LIN {X 0,Y 466.661,Z 585.899,A -85,B 0,C 180,E1 -7456.944,E2 -7456.944} C_VEL
LIN {X 0,Y 466.788,Z 583.643,A -85,B 0,C 180,E1 -7458.141,E2 -7458.141} C_VEL
LIN {X 0,Y 466.923,Z 579.745,A -85,B 0,C 180,E1 -7459.594,E2 -7459.594} C_VEL
LIN {X 0,Y 467.085,Z 575.044,A -85,B 0,C 180,E1 -7460.91,E2 -7460.91} C_VEL
LIN {X 0,Y 467.42,Z 568.051,A -85,B 0,C 180,E1 -7462.424,E2 -7462.424} C_VEL
LIN {X 0,Y 467.776,Z 560.313,A -85,B 0,C 180,E1 -7463.747,E2 -7463.747} C_VEL
LIN {X 0,Y 468.215,Z 550.713,A -85,B 0,C 180,E1 -7465.049,E2 -7465.049} C_VEL
LIN {X 0,Y 468.714,Z 540.809,A -85,B 0,C 180,E1 -7466.131,E2 -7466.131} C_VEL
LIN {X 0,Y 469.163,Z 529.664,A -85,B 0,C 180,E1 -7467.102,E2 -7467.102} C_VEL
LIN {X 0,Y 469.668,Z 518.712,A -85,B 0,C 180,E1 -7467.856,E2 -7467.856} C_VEL
LIN {X 0,Y 470.068,Z 506.643,A -85,B 0,C 180,E1 -7468.501,E2 -7468.501} C_VEL
LIN {X 0,Y 470.446,Z 493.985,A -85,B 0,C 180,E1 -7468.984,E2 -7468.984} C_VEL
LIN {X 0,Y 470.619,Z 481.549,A -85,B 0,C 180,E1 -7469.291,E2 -7469.291} C_VEL
LIN {X 0,Y 471.254,Z 391.992,A -85,B 0,C 180,E1 -7470.675,E2 -7470.675} C_VEL
LIN {X 0,Y 468.455,Z 378.274,A -85,B 0,C 180,E1 -7470.994,E2 -7470.994} C_VEL
LIN {X 0,Y 468.774,Z 369.227,A -85,B 0,C 180,E1 -7473.008,E2 -7473.008} C_VEL
LIN {X 0,Y 467.628,Z 363.237,A -85,B 0,C 180,E1 -7474.471,E2 -7474.471} C_VEL
LIN {X 0,Y 467.667,Z 363.231,A -85,B 0,C 180,E1 -7476.905,E2 -7476.905} C_VEL
LIN {X 0,Y 467.668,Z 363.233,A -85,B 0,C 180,E1 -7479.515,E2 -7479.515} C_VEL
LIN {X 0,Y 467.659,Z 363.227,A -85,B 0,C 180,E1 -7482.357,E2 -7482.357} C_VEL
LIN {X 0,Y 467.654,Z 363.229,A -85,B 0,C 180,E1 -7485.885,E2 -7485.885} C_VEL
LIN {X 0,Y 467.627,Z 363.239,A -85,B 0,C 180,E1 -7489.307,E2 -7489.307} C_VEL
LIN {X 0,Y 467.54,Z 363.242,A -85,B 0,C 180,E1 -7492.073,E2 -7492.073} C_VEL
LIN {X 0,Y 467.607,Z 363.237,A -85,B 0,C 180,E1 -7494.886,E2 -7494.886} C_VEL
LIN {X 0,Y 467.622,Z 363.233,A -85,B 0,C 180,E1 -7497.768,E2 -7497.768} C_VEL
LIN {X 0,Y 467.577,Z 363.243,A -85,B 0,C 180,E1 -7501.046,E2 -7501.046} C_VEL
LIN {X 0,Y 467.591,Z 363.235,A -85,B 0,C 180,E1 -7504.242,E2 -7504.242} C_VEL
LIN {X 0,Y 467.551,Z 363.247,A -85,B 0,C 180,E1 -7507.186,E2 -7507.186} C_VEL
LIN {X 0,Y 467.577,Z 363.237,A -85,B 0,C 180,E1 -7510.264,E2 -7510.264} C_VEL
LIN {X 0,Y 467.585,Z 363.238,A -85,B 0,C 180,E1 -7512.566,E2 -7512.566} C_VEL
LIN {X 0,Y 467.569,Z 363.246,A -85,B 0,C 180,E1 -7515.052,E2 -7515.052} C_VEL
LIN {X 0,Y 467.586,Z 363.238,A -85,B 0,C 180,E1 -7517.439,E2 -7517.439} C_VEL
LIN {X 0,Y 467.581,Z 363.243,A -85,B 0,C 180,E1 -7520.855,E2 -7520.855} C_VEL
LIN {X 0,Y 467.558,Z 363.24,A -85,B 0,C 180,E1 -7524.259,E2 -7524.259} C_VEL
LIN {X 0,Y 467.577,Z 363.24,A -85,B 0,C 180,E1 -7527.32,E2 -7527.32} C_VEL
LIN {X 0,Y 467.564,Z 363.244,A -85,B 0,C 180,E1 -7530.666,E2 -7530.666} C_VEL
LIN {X 0,Y 467.621,Z 363.235,A -85,B 0,C 180,E1 -7533.2,E2 -7533.2} C_VEL
LIN {X 0,Y 467.586,Z 363.24,A -85,B 0,C 180,E1 -7536.467,E2 -7536.467} C_VEL
LIN {X 0,Y 467.616,Z 363.232,A -85,B 0,C 180,E1 -7539.777,E2 -7539.777} C_VEL
LIN {X 0,Y 467.602,Z 363.239,A -85,B 0,C 180,E1 -7542.506,E2 -7542.506} C_VEL
LIN {X 0,Y 467.598,Z 363.236,A -85,B 0,C 180,E1 -7545.196,E2 -7545.196} C_VEL
LIN {X 0,Y 467.648,Z 363.228,A -85,B 0,C 180,E1 -7547.854,E2 -7547.854} C_VEL
LIN {X 0,Y 467.674,Z 363.225,A -85,B 0,C 180,E1 -7551.357,E2 -7551.357} C_VEL
LIN {X 0,Y 467.738,Z 363.218,A -85,B 0,C 180,E1 -7553.962,E2 -7553.962} C_VEL
LIN {X 0,Y 467.852,Z 363.203,A -85,B 0,C 180,E1 -7557.417,E2 -7557.417} C_VEL
LIN {X 0,Y 467.873,Z 363.202,A -85,B 0,C 180,E1 -7560,E2 -7560} C_VEL
LIN {X 0,Y 467.851,Z 363.21,A -85,B 0,C 180,E1 -7562.583,E2 -7562.583} C_VEL
LIN {X 0,Y 467.734,Z 363.22,A -85,B 0,C 180,E1 -7566.037,E2 -7566.037} C_VEL
LIN {X 0,Y 467.673,Z 363.23,A -85,B 0,C 180,E1 -7568.643,E2 -7568.643} C_VEL
LIN {X 0,Y 467.647,Z 363.233,A -85,B 0,C 180,E1 -7572.146,E2 -7572.146} C_VEL
LIN {X 0,Y 467.657,Z 363.229,A -85,B 0,C 180,E1 -7575.893,E2 -7575.893} C_VEL
LIN {X 0,Y 467.615,Z 363.232,A -85,B 0,C 180,E1 -7579.308,E2 -7579.308} C_VEL
LIN {X 0,Y 467.528,Z 363.248,A -85,B 0,C 180,E1 -7582.074,E2 -7582.074} C_VEL
LIN {X 0,Y 467.595,Z 363.236,A -85,B 0,C 180,E1 -7584.888,E2 -7584.888} C_VEL
LIN {X 0,Y 467.621,Z 363.234,A -85,B 0,C 180,E1 -7587.769,E2 -7587.769} C_VEL
LIN {X 0,Y 467.565,Z 363.238,A -85,B 0,C 180,E1 -7591.046,E2 -7591.046} C_VEL
LIN {X 0,Y 467.584,Z 363.243,A -85,B 0,C 180,E1 -7594.243,E2 -7594.243} C_VEL
LIN {X 0,Y 467.546,Z 363.241,A -85,B 0,C 180,E1 -7597.188,E2 -7597.188} C_VEL
LIN {X 0,Y 467.592,Z 363.241,A -85,B 0,C 180,E1 -7600.263,E2 -7600.263} C_VEL
LIN {X 0,Y 467.614,Z 363.234,A -85,B 0,C 180,E1 -7602.572,E2 -7602.572} C_VEL
LIN {X 0,Y 467.566,Z 363.238,A -85,B 0,C 180,E1 -7605.054,E2 -7605.054} C_VEL
LIN {X 0,Y 467.585,Z 363.238,A -85,B 0,C 180,E1 -7607.441,E2 -7607.441} C_VEL
LIN {X 0,Y 467.621,Z 363.231,A -85,B 0,C 180,E1 -7610.86,E2 -7610.86} C_VEL
LIN {X 0,Y 467.561,Z 363.243,A -85,B 0,C 180,E1 -7614.261,E2 -7614.261} C_VEL
LIN {X 0,Y 467.581,Z 363.238,A -85,B 0,C 180,E1 -7617.321,E2 -7617.321} C_VEL
LIN {X 0,Y 467.578,Z 363.242,A -85,B 0,C 180,E1 -7620.666,E2 -7620.666} C_VEL
LIN {X 0,Y 467.666,Z 363.405,A -85,B 0,C 180,E1 -7623.445,E2 -7623.445} C_VEL
LIN {X 0,Y 470.093,Z 376.061,A -85,B 0,C 180,E1 -7625.779,E2 -7625.779} C_VEL
LIN {X 0,Y 469.334,Z 392.226,A -85,B 0,C 180,E1 -7628.532,E2 -7628.532} C_VEL
LIN {X 0,Y 468.677,Z 409.488,A -85,B 0,C 180,E1 -7631.437,E2 -7631.437} C_VEL
LIN {X 0,Y 468.279,Z 418.901,A -85,B 0,C 180,E1 -7633.007,E2 -7633.007} C_VEL
LIN {X 0,Y 471.13,Z 438.244,A -85,B 0,C 180,E1 -7633.413,E2 -7633.413} C_VEL
LIN {X 0,Y 470.44,Z 528.202,A -85,B 0,C 180,E1 -7634.817,E2 -7634.817} C_VEL
LIN {X 0,Y 470.054,Z 541.256,A -85,B 0,C 180,E1 -7635.193,E2 -7635.193} C_VEL
LIN {X 0,Y 469.629,Z 553.327,A -85,B 0,C 180,E1 -7635.705,E2 -7635.705} C_VEL
LIN {X 0,Y 469.159,Z 564.727,A -85,B 0,C 180,E1 -7636.354,E2 -7636.354} C_VEL
LIN {X 0,Y 468.609,Z 576.235,A -85,B 0,C 180,E1 -7637.2,E2 -7637.2} C_VEL
LIN {X 0,Y 468.208,Z 587.031,A -85,B 0,C 180,E1 -7638.199,E2 -7638.199} C_VEL
LIN {X 0,Y 467.767,Z 595.658,A -85,B 0,C 180,E1 -7639.175,E2 -7639.175} C_VEL
LIN {X 0,Y 467.397,Z 603.616,A -85,B 0,C 180,E1 -7640.261,E2 -7640.261} C_VEL
LIN {X 0,Y 467.103,Z 611.392,A -85,B 0,C 180,E1 -7641.565,E2 -7641.565} C_VEL
LIN {X 0,Y 466.858,Z 618.538,A -85,B 0,C 180,E1 -7643.083,E2 -7643.083} C_VEL
LIN {X 0,Y 466.762,Z 623.297,A -85,B 0,C 180,E1 -7644.384,E2 -7644.384} C_VEL
LIN {X 0,Y 466.658,Z 626.931,A -85,B 0,C 180,E1 -7645.682,E2 -7645.682} C_VEL
LIN {X 0,Y 466.697,Z 628.81,A -85,B 0,C 180,E1 -7646.547,E2 -7646.547} C_VEL
LIN {X 0,Y 466.68,Z 630.217,A -85,B 0,C 180,E1 -7647.411,E2 -7647.411} C_VEL
LIN {X 0,Y 466.661,Z 631.218,A -85,B 0,C 180,E1 -7648.274,E2 -7648.274} C_VEL
LIN {X 0,Y 466.6,Z 632.044,A -85,B 0,C 180,E1 -7650,E2 -7650} C_VEL
LIN {X 0,Y 466.62,Z 631.827,A -85,B 0,C 180,E1 -7650.863,E2 -7650.863} C_VEL
LIN {X 0,Y 466.661,Z 631.216,A -85,B 0,C 180,E1 -7651.726,E2 -7651.726} C_VEL
LIN {X 0,Y 466.68,Z 630.212,A -85,B 0,C 180,E1 -7652.589,E2 -7652.589} C_VEL
LIN {X 0,Y 466.697,Z 628.807,A -85,B 0,C 180,E1 -7653.453,E2 -7653.453} C_VEL
LIN {X 0,Y 466.69,Z 625.849,A -85,B 0,C 180,E1 -7654.751,E2 -7654.751} C_VEL
LIN {X 0,Y 466.751,Z 621.85,A -85,B 0,C 180,E1 -7656.05,E2 -7656.05} C_VEL
LIN {X 0,Y 466.942,Z 615.716,A -85,B 0,C 180,E1 -7657.568,E2 -7657.568} C_VEL
LIN {X 0,Y 467.15,Z 609.018,A -85,B 0,C 180,E1 -7658.87,E2 -7658.87} C_VEL
LIN {X 0,Y 467.494,Z 600.717,A -85,B 0,C 180,E1 -7660.174,E2 -7660.174} C_VEL
LIN {X 0,Y 467.967,Z 592.229,A -85,B 0,C 180,E1 -7661.258,E2 -7661.258} C_VEL
LIN {X 0,Y 468.439,Z 582.273,A -85,B 0,C 180,E1 -7662.296,E2 -7662.296} C_VEL
LIN {X 0,Y 468.875,Z 571.396,A -85,B 0,C 180,E1 -7663.213,E2 -7663.213} C_VEL
LIN {X 0,Y 469.435,Z 560.072,A -85,B 0,C 180,E1 -7663.969,E2 -7663.969} C_VEL
LIN {X 0,Y 469.907,Z 548.54,A -85,B 0,C 180,E1 -7664.563,E2 -7664.563} C_VEL
LIN {X 0,Y 470.36,Z 535.317,A -85,B 0,C 180,E1 -7665.047,E2 -7665.047} C_VEL
LIN {X 0,Y 470.643,Z 522.537,A -85,B 0,C 180,E1 -7665.342,E2 -7665.342} C_VEL
LIN {X 0,Y 471.202,Z 437.855,A -85,B 0,C 180,E1 -7666.654,E2 -7666.654} C_VEL
LIN {X 0,Y 468.339,Z 418.514,A -85,B 0,C 180,E1 -7667.095,E2 -7667.095} C_VEL
LIN {X 0,Y 469.097,Z 400.424,A -85,B 0,C 180,E1 -7670.156,E2 -7670.156} C_VEL
LIN {X 0,Y 469.966,Z 381.889,A -85,B 0,C 180,E1 -7673.346,E2 -7673.346} C_VEL
LIN {X 0,Y 470.14,Z 375.734,A -85,B 0,C 180,E1 -7674.428,E2 -7674.428} C_VEL
LIN {X 0,Y 467.686,Z 363.229,A -85,B 0,C 180,E1 -7676.851,E2 -7676.851} C_VEL
LIN {X 0,Y 467.587,Z 363.241,A -85,B 0,C 180,E1 -7679.735,E2 -7679.735} C_VEL
LIN {X 0,Y 467.582,Z 363.238,A -85,B 0,C 180,E1 -7682.758,E2 -7682.758} C_VEL
LIN {X 0,Y 467.555,Z 363.248,A -85,B 0,C 180,E1 -7685.889,E2 -7685.889} C_VEL
LIN {X 0,Y 467.621,Z 363.231,A -85,B 0,C 180,E1 -7689.14,E2 -7689.14} C_VEL
LIN {X 0,Y 467.582,Z 363.237,A -85,B 0,C 180,E1 -7692.566,E2 -7692.566} C_VEL
LIN {X 0,Y 467.566,Z 363.239,A -85,B 0,C 180,E1 -7695.052,E2 -7695.052} C_VEL
LIN {X 0,Y 467.619,Z 363.236,A -85,B 0,C 180,E1 -7697.443,E2 -7697.443} C_VEL
LIN {X 0,Y 467.613,Z 363.233,A -85,B 0,C 180,E1 -7700.858,E2 -7700.858} C_VEL
LIN {X 0,Y 467.557,Z 363.243,A -85,B 0,C 180,E1 -7704.26,E2 -7704.26} C_VEL
LIN {X 0,Y 467.576,Z 363.238,A -85,B 0,C 180,E1 -7707.32,E2 -7707.32} C_VEL
LIN {X 0,Y 467.57,Z 363.236,A -85,B 0,C 180,E1 -7710.665,E2 -7710.665} C_VEL
LIN {X 0,Y 467.62,Z 363.234,A -85,B 0,C 180,E1 -7713.2,E2 -7713.2} C_VEL
LIN {X 0,Y 467.584,Z 363.237,A -85,B 0,C 180,E1 -7716.468,E2 -7716.468} C_VEL
LIN {X 0,Y 467.615,Z 363.239,A -85,B 0,C 180,E1 -7719.777,E2 -7719.777} C_VEL
LIN {X 0,Y 467.6,Z 363.23,A -85,B 0,C 180,E1 -7722.507,E2 -7722.507} C_VEL
LIN {X 0,Y 467.6,Z 363.238,A -85,B 0,C 180,E1 -7725.196,E2 -7725.196} C_VEL
LIN {X 0,Y 467.647,Z 363.23,A -85,B 0,C 180,E1 -7727.854,E2 -7727.854} C_VEL
LIN {X 0,Y 467.673,Z 363.23,A -85,B 0,C 180,E1 -7731.357,E2 -7731.357} C_VEL
LIN {X 0,Y 467.735,Z 363.219,A -85,B 0,C 180,E1 -7733.963,E2 -7733.963} C_VEL
LIN {X 0,Y 467.852,Z 363.205,A -85,B 0,C 180,E1 -7737.417,E2 -7737.417} C_VEL
LIN {X 0,Y 467.873,Z 363.202,A -85,B 0,C 180,E1 -7740,E2 -7740} C_VEL
LIN {X 0,Y 467.853,Z 363.199,A -85,B 0,C 180,E1 -7742.583,E2 -7742.583} C_VEL
LIN {X 0,Y 467.739,Z 363.216,A -85,B 0,C 180,E1 -7746.038,E2 -7746.038} C_VEL
LIN {X 0,Y 467.674,Z 363.225,A -85,B 0,C 180,E1 -7748.643,E2 -7748.643} C_VEL
LIN {X 0,Y 467.648,Z 363.224,A -85,B 0,C 180,E1 -7752.146,E2 -7752.146} C_VEL
LIN {X 0,Y 467.631,Z 363.229,A -85,B 0,C 180,E1 -7755.696,E2 -7755.696} C_VEL
LIN {X 0,Y 467.61,Z 363.238,A -85,B 0,C 180,E1 -7758.765,E2 -7758.765} C_VEL
LIN {X 0,Y 467.603,Z 363.24,A -85,B 0,C 180,E1 -7761.278,E2 -7761.278} C_VEL
LIN {X 0,Y 467.568,Z 363.235,A -85,B 0,C 180,E1 -7763.944,E2 -7763.944} C_VEL
LIN {X 0,Y 467.622,Z 363.238,A -85,B 0,C 180,E1 -7766.8,E2 -7766.8} C_VEL
LIN {X 0,Y 467.548,Z 363.241,A -85,B 0,C 180,E1 -7769.739,E2 -7769.739} C_VEL
LIN {X 0,Y 467.579,Z 363.243,A -85,B 0,C 180,E1 -7772.759,E2 -7772.759} C_VEL
LIN {X 0,Y 467.552,Z 363.241,A -85,B 0,C 180,E1 -7775.89,E2 -7775.89} C_VEL
LIN {X 0,Y 467.609,Z 363.237,A -85,B 0,C 180,E1 -7779.143,E2 -7779.143} C_VEL
LIN {X 0,Y 467.616,Z 363.234,A -85,B 0,C 180,E1 -7782.572,E2 -7782.572} C_VEL
LIN {X 0,Y 467.565,Z 363.242,A -85,B 0,C 180,E1 -7786.178,E2 -7786.178} C_VEL
LIN {X 0,Y 467.581,Z 363.244,A -85,B 0,C 180,E1 -7788.724,E2 -7788.724} C_VEL
LIN {X 0,Y 467.567,Z 363.247,A -85,B 0,C 180,E1 -7791.957,E2 -7791.957} C_VEL
LIN {X 0,Y 467.584,Z 363.359,A -85,B 0,C 180,E1 -7793.447,E2 -7793.447} C_VEL
LIN {X 0,Y 468.911,Z 370.963,A -85,B 0,C 180,E1 -7795.283,E2 -7795.283} C_VEL
LIN {X 0,Y 468.587,Z 378.596,A -85,B 0,C 180,E1 -7797.004,E2 -7797.004} C_VEL
LIN {X 0,Y 471.51,Z 392.271,A -85,B 0,C 180,E1 -7797.341,E2 -7797.341} C_VEL
LIN {X 0,Y 470.71,Z 485.56,A -85,B 0,C 180,E1 -7798.809,E2 -7798.809} C_VEL
LIN {X 0,Y 470.376,Z 499.472,A -85,B 0,C 180,E1 -7799.221,E2 -7799.221} C_VEL
LIN {X 0,Y 470.126,Z 509.899,A -85,B 0,C 180,E1 -7799.676,E2 -7799.676} C_VEL
LIN {X 0,Y 469.281,Z 515.36,A -85,B 0,C 180,E1 -7799.935,E2 -7799.935} C_VEL
LIN {X 0,Y 466.173,Z 524.081,A -85,B 0,C 180,E1 -7800.375,E2 -7800.375} C_VEL
LIN {X 0,Y 463.03,Z 532.395,A -85,B 0,C 180,E1 -7800.911,E2 -7800.911} C_VEL
LIN {X 0,Y 462.133,Z 537.212,A -85,B 0,C 180,E1 -7801.316,E2 -7801.316} C_VEL
LIN {X 0,Y 461.567,Z 547.235,A -85,B 0,C 180,E1 -7802.34,E2 -7802.34} C_VEL
LIN {X 0,Y 461.087,Z 556.615,A -85,B 0,C 180,E1 -7803.524,E2 -7803.524} C_VEL
LIN {X 0,Y 460.653,Z 564.295,A -85,B 0,C 180,E1 -7804.712,E2 -7804.712} C_VEL
LIN {X 0,Y 460.305,Z 571.371,A -85,B 0,C 180,E1 -7806.071,E2 -7806.071} C_VEL
LIN {X 0,Y 460.007,Z 577.418,A -85,B 0,C 180,E1 -7807.546,E2 -7807.546} C_VEL
LIN {X 0,Y 459.827,Z 581.418,A -85,B 0,C 180,E1 -7808.802,E2 -7808.802} C_VEL
LIN {X 0,Y 459.627,Z 585.046,A -85,B 0,C 180,E1 -7810.343,E2 -7810.343} C_VEL
LIN {X 0,Y 459.552,Z 586.854,A -85,B 0,C 180,E1 -7811.475,E2 -7811.475} C_VEL
LIN {X 0,Y 459.455,Z 588.29,A -85,B 0,C 180,E1 -7813.105,E2 -7813.105} C_VEL
LIN {X 0,Y 459.504,Z 588.432,A -85,B 0,C 180,E1 -7814.489,E2 -7814.489} C_VEL
LIN {X 0,Y 459.503,Z 587.632,A -85,B 0,C 180,E1 -7815.835,E2 -7815.835} C_VEL
LIN {X 0,Y 459.568,Z 586.585,A -85,B 0,C 180,E1 -7816.739,E2 -7816.739} C_VEL
LIN {X 0,Y 459.7,Z 584.19,A -85,B 0,C 180,E1 -7818.085,E2 -7818.085} C_VEL
LIN {X 0,Y 459.824,Z 580.778,A -85,B 0,C 180,E1 -7819.432,E2 -7819.432} C_VEL
LIN {X 0,Y 460.006,Z 576.286,A -85,B 0,C 180,E1 -7820.769,E2 -7820.769} C_VEL
LIN {X 0,Y 460.314,Z 570.574,A -85,B 0,C 180,E1 -7822.102,E2 -7822.102} C_VEL
LIN {X 0,Y 460.59,Z 563.441,A -85,B 0,C 180,E1 -7823.429,E2 -7823.429} C_VEL
LIN {X 0,Y 461.052,Z 554.563,A -85,B 0,C 180,E1 -7824.753,E2 -7824.753} C_VEL
LIN {X 0,Y 461.515,Z 545.469,A -85,B 0,C 180,E1 -7825.852,E2 -7825.852} C_VEL
LIN {X 0,Y 462.053,Z 535.361,A -85,B 0,C 180,E1 -7826.839,E2 -7826.839} C_VEL
LIN {X 0,Y 462.54,Z 524.184,A -85,B 0,C 180,E1 -7827.714,E2 -7827.714} C_VEL
LIN {X 0,Y 463.041,Z 511.602,A -85,B 0,C 180,E1 -7828.478,E2 -7828.478} C_VEL
LIN {X 0,Y 463.381,Z 498.597,A -85,B 0,C 180,E1 -7829.05,E2 -7829.05} C_VEL
LIN {X 0,Y 463.651,Z 485.695,A -85,B 0,C 180,E1 -7829.43,E2 -7829.43} C_VEL
LIN {X 0,Y 464.534,Z 398.268,A -85,B 0,C 180,E1 -7830.813,E2 -7830.813} C_VEL
LIN {X 0,Y 464.318,Z 392.241,A -85,B 0,C 180,E1 -7830.916,E2 -7830.916} C_VEL
LIN {X 0,Y 461.51,Z 378.564,A -85,B 0,C 180,E1 -7831.241,E2 -7831.241} C_VEL
LIN {X 0,Y 461.787,Z 370.5,A -85,B 0,C 180,E1 -7833.053,E2 -7833.053} C_VEL
LIN {X 0,Y 460.589,Z 364.114,A -85,B 0,C 180,E1 -7834.595,E2 -7834.595} C_VEL
LIN {X 0,Y 460.674,Z 364.105,A -85,B 0,C 180,E1 -7837.412,E2 -7837.412} C_VEL
LIN {X 0,Y 460.584,Z 364.108,A -85,B 0,C 180,E1 -7840.551,E2 -7840.551} C_VEL
LIN {X 0,Y 460.554,Z 364.118,A -85,B 0,C 180,E1 -7843.232,E2 -7843.232} C_VEL
LIN {X 0,Y 460.605,Z 364.106,A -85,B 0,C 180,E1 -7845.997,E2 -7845.997} C_VEL
LIN {X 0,Y 460.575,Z 364.112,A -85,B 0,C 180,E1 -7848.901,E2 -7848.901} C_VEL
LIN {X 0,Y 460.52,Z 364.121,A -85,B 0,C 180,E1 -7851.485,E2 -7851.485} C_VEL
LIN {X 0,Y 460.546,Z 364.113,A -85,B 0,C 180,E1 -7854.331,E2 -7854.331} C_VEL
LIN {X 0,Y 460.576,Z 364.117,A -85,B 0,C 180,E1 -7857.243,E2 -7857.243} C_VEL
LIN {X 0,Y 460.517,Z 364.116,A -85,B 0,C 180,E1 -7860.239,E2 -7860.239} C_VEL
LIN {X 0,Y 460.531,Z 364.121,A -85,B 0,C 180,E1 -7863.324,E2 -7863.324} C_VEL
LIN {X 0,Y 460.48,Z 364.122,A -85,B 0,C 180,E1 -7866.528,E2 -7866.528} C_VEL
LIN {X 0,Y 460.557,Z 364.112,A -85,B 0,C 180,E1 -7869.859,E2 -7869.859} C_VEL
LIN {X 0,Y 460.512,Z 364.123,A -85,B 0,C 180,E1 -7872.899,E2 -7872.899} C_VEL
LIN {X 0,Y 460.521,Z 364.116,A -85,B 0,C 180,E1 -7875.828,E2 -7875.828} C_VEL
LIN {X 0,Y 460.531,Z 364.123,A -85,B 0,C 180,E1 -7878.988,E2 -7878.988} C_VEL
LIN {X 0,Y 460.528,Z 364.119,A -85,B 0,C 180,E1 -7881.267,E2 -7881.267} C_VEL
LIN {X 0,Y 460.509,Z 364.121,A -85,B 0,C 180,E1 -7884.554,E2 -7884.554} C_VEL
LIN {X 0,Y 460.527,Z 364.115,A -85,B 0,C 180,E1 -7887.715,E2 -7887.715} C_VEL
LIN {X 0,Y 460.534,Z 364.121,A -85,B 0,C 180,E1 -7890.768,E2 -7890.768} C_VEL
LIN {X 0,Y 460.562,Z 364.111,A -85,B 0,C 180,E1 -7893.734,E2 -7893.734} C_VEL
LIN {X 0,Y 460.539,Z 364.12,A -85,B 0,C 180,E1 -7896.623,E2 -7896.623} C_VEL
LIN {X 0,Y 460.545,Z 364.114,A -85,B 0,C 180,E1 -7899.452,E2 -7899.452} C_VEL
LIN {X 0,Y 460.552,Z 364.114,A -85,B 0,C 180,E1 -7902.23,E2 -7902.23} C_VEL
LIN {X 0,Y 460.557,Z 364.116,A -85,B 0,C 180,E1 -7904.964,E2 -7904.964} C_VEL
LIN {X 0,Y 460.601,Z 364.106,A -85,B 0,C 180,E1 -7907.665,E2 -7907.665} C_VEL
LIN {X 0,Y 460.621,Z 364.105,A -85,B 0,C 180,E1 -7911.223,E2 -7911.223} C_VEL
LIN {X 0,Y 460.704,Z 364.094,A -85,B 0,C 180,E1 -7913.87,E2 -7913.87} C_VEL
LIN {X 0,Y 460.817,Z 364.079,A -85,B 0,C 180,E1 -7917.377,E2 -7917.377} C_VEL
LIN {X 0,Y 460.843,Z 364.078,A -85,B 0,C 180,E1 -7920,E2 -7920} C_VEL
LIN {X 0,Y 460.816,Z 364.086,A -85,B 0,C 180,E1 -7922.622,E2 -7922.622} C_VEL
LIN {X 0,Y 460.7,Z 364.097,A -85,B 0,C 180,E1 -7926.13,E2 -7926.13} C_VEL
LIN {X 0,Y 460.62,Z 364.107,A -85,B 0,C 180,E1 -7928.776,E2 -7928.776} C_VEL
LIN {X 0,Y 460.604,Z 364.113,A -85,B 0,C 180,E1 -7932.445,E2 -7932.445} C_VEL
LIN {X 0,Y 460.613,Z 364.108,A -85,B 0,C 180,E1 -7936.007,E2 -7936.007} C_VEL
LIN {X 0,Y 460.561,Z 364.112,A -85,B 0,C 180,E1 -7939.616,E2 -7939.616} C_VEL
LIN {X 0,Y 460.504,Z 364.124,A -85,B 0,C 180,E1 -7942.429,E2 -7942.429} C_VEL
LIN {X 0,Y 460.561,Z 364.114,A -85,B 0,C 180,E1 -7945.803,E2 -7945.803} C_VEL
LIN {X 0,Y 460.551,Z 364.12,A -85,B 0,C 180,E1 -7948.233,E2 -7948.233} C_VEL
LIN {X 0,Y 460.518,Z 364.116,A -85,B 0,C 180,E1 -7951.284,E2 -7951.284} C_VEL
LIN {X 0,Y 460.528,Z 364.118,A -85,B 0,C 180,E1 -7954.507,E2 -7954.507} C_VEL
LIN {X 0,Y 460.525,Z 364.118,A -85,B 0,C 180,E1 -7957.621,E2 -7957.621} C_VEL
LIN {X 0,Y 460.555,Z 364.117,A -85,B 0,C 180,E1 -7960.273,E2 -7960.273} C_VEL
LIN {X 0,Y 460.52,Z 364.117,A -85,B 0,C 180,E1 -7963.373,E2 -7963.373} C_VEL
LIN {X 0,Y 460.495,Z 364.12,A -85,B 0,C 180,E1 -7966.625,E2 -7966.625} C_VEL
LIN {X 0,Y 460.559,Z 364.116,A -85,B 0,C 180,E1 -7969.728,E2 -7969.728} C_VEL
LIN {X 0,Y 460.526,Z 364.117,A -85,B 0,C 180,E1 -7972.52,E2 -7972.52} C_VEL
LIN {X 0,Y 460.547,Z 364.117,A -85,B 0,C 180,E1 -7975.625,E2 -7975.625} C_VEL
LIN {X 0,Y 460.535,Z 364.114,A -85,B 0,C 180,E1 -7978.745,E2 -7978.745} C_VEL
LIN {X 0,Y 460.558,Z 364.121,A -85,B 0,C 180,E1 -7981.768,E2 -7981.768} C_VEL
LIN {X 0,Y 460.644,Z 364.3,A -85,B 0,C 180,E1 -7983.252,E2 -7983.252} C_VEL
LIN {X 0,Y 463.082,Z 376.75,A -85,B 0,C 180,E1 -7985.588,E2 -7985.588} C_VEL
LIN {X 0,Y 462.542,Z 390.357,A -85,B 0,C 180,E1 -7987.949,E2 -7987.949} C_VEL
LIN {X 0,Y 461.664,Z 410.286,A -85,B 0,C 180,E1 -7991.356,E2 -7991.356} C_VEL
LIN {X 0,Y 461.3,Z 418.542,A -85,B 0,C 180,E1 -7992.755,E2 -7992.755} C_VEL
LIN {X 0,Y 464.278,Z 438.909,A -85,B 0,C 180,E1 -7993.192,E2 -7993.192} C_VEL
LIN {X 0,Y 463.597,Z 527.285,A -85,B 0,C 180,E1 -7994.588,E2 -7994.588} C_VEL
LIN {X 0,Y 463.173,Z 540.53,A -85,B 0,C 180,E1 -7994.967,E2 -7994.967} C_VEL
LIN {X 0,Y 462.686,Z 553.825,A -85,B 0,C 180,E1 -7995.542,E2 -7995.542} C_VEL
LIN {X 0,Y 462.156,Z 565.788,A -85,B 0,C 180,E1 -7996.255,E2 -7996.255} C_VEL
LIN {X 0,Y 461.561,Z 577.959,A -85,B 0,C 180,E1 -7997.193,E2 -7997.193} C_VEL
LIN {X 0,Y 461.171,Z 587.634,A -85,B 0,C 180,E1 -7998.128,E2 -7998.128} C_VEL
LIN {X 0,Y 460.655,Z 596.928,A -85,B 0,C 180,E1 -7999.229,E2 -7999.229} C_VEL
LIN {X 0,Y 460.202,Z 605.962,A -85,B 0,C 180,E1 -8000.551,E2 -8000.551} C_VEL
LIN {X 0,Y 459.935,Z 613.242,A -85,B 0,C 180,E1 -8001.875,E2 -8001.875} C_VEL
LIN {X 0,Y 459.742,Z 619.342,A -85,B 0,C 180,E1 -8003.273,E2 -8003.273} C_VEL
LIN {X 0,Y 459.668,Z 624.26,A -85,B 0,C 180,E1 -8004.737,E2 -8004.737} C_VEL
LIN {X 0,Y 459.573,Z 626.574,A -85,B 0,C 180,E1 -8005.615,E2 -8005.615} C_VEL
LIN {X 0,Y 459.595,Z 628.459,A -85,B 0,C 180,E1 -8006.493,E2 -8006.493} C_VEL
LIN {X 0,Y 459.601,Z 629.874,A -85,B 0,C 180,E1 -8007.371,E2 -8007.371} C_VEL
LIN {X 0,Y 459.553,Z 631.49,A -85,B 0,C 180,E1 -8009.124,E2 -8009.124} C_VEL
LIN {X 0,Y 459.532,Z 631.711,A -85,B 0,C 180,E1 -8010,E2 -8010} C_VEL
LIN {X 0,Y 459.553,Z 631.499,A -85,B 0,C 180,E1 -8010.876,E2 -8010.876} C_VEL
LIN {X 0,Y 459.601,Z 629.889,A -85,B 0,C 180,E1 -8012.629,E2 -8012.629} C_VEL
LIN {X 0,Y 459.594,Z 628.487,A -85,B 0,C 180,E1 -8013.507,E2 -8013.507} C_VEL
LIN {X 0,Y 459.621,Z 625.538,A -85,B 0,C 180,E1 -8014.824,E2 -8014.824} C_VEL
LIN {X 0,Y 459.714,Z 620.523,A -85,B 0,C 180,E1 -8016.431,E2 -8016.431} C_VEL
LIN {X 0,Y 459.89,Z 614.415,A -85,B 0,C 180,E1 -8017.905,E2 -8017.905} C_VEL
LIN {X 0,Y 460.171,Z 607.504,A -85,B 0,C 180,E1 -8019.228,E2 -8019.228} C_VEL
LIN {X 0,Y 460.562,Z 598.881,A -85,B 0,C 180,E1 -8020.551,E2 -8020.551} C_VEL
LIN {X 0,Y 461.055,Z 590.043,A -85,B 0,C 180,E1 -8021.652,E2 -8021.652} C_VEL
LIN {X 0,Y 461.546,Z 579.462,A -85,B 0,C 180,E1 -8022.728,E2 -8022.728} C_VEL
LIN {X 0,Y 462.108,Z 568.281,A -85,B 0,C 180,E1 -8023.634,E2 -8023.634} C_VEL
LIN {X 0,Y 462.661,Z 556.096,A -85,B 0,C 180,E1 -8024.403,E2 -8024.403} C_VEL
LIN {X 0,Y 463.26,Z 543.351,A -85,B 0,C 180,E1 -8025.002,E2 -8025.002} C_VEL
LIN {X 0,Y 463.652,Z 530.664,A -85,B 0,C 180,E1 -8025.41,E2 -8025.41} C_VEL
LIN {X 0,Y 463.9,Z 512.82,A -85,B 0,C 180,E1 -8025.74,E2 -8025.74} C_VEL
LIN {X 0,Y 464.405,Z 438.362,A -85,B 0,C 180,E1 -8026.912,E2 -8026.912} C_VEL
LIN {X 0,Y 461.378,Z 418.292,A -85,B 0,C 180,E1 -8027.363,E2 -8027.363} C_VEL
LIN {X 0,Y 462.137,Z 401.558,A -85,B 0,C 180,E1 -8030.241,E2 -8030.241} C_VEL
LIN {X 0,Y 463.05,Z 383.077,A -85,B 0,C 180,E1 -8033.478,E2 -8033.478} C_VEL
LIN {X 0,Y 463.281,Z 377.527,A -85,B 0,C 180,E1 -8034.466,E2 -8034.466} C_VEL
LIN {X 0,Y 460.997,Z 365.937,A -85,B 0,C 180,E1 -8036.726,E2 -8036.726} C_VEL
LIN {X 0,Y 460.656,Z 364.105,A -85,B 0,C 180,E1 -8037.115,E2 -8037.115} C_VEL
LIN {X 0,Y 460.527,Z 364.124,A -85,B 0,C 180,E1 -8040.238,E2 -8040.238} C_VEL
LIN {X 0,Y 460.528,Z 364.116,A -85,B 0,C 180,E1 -8043.324,E2 -8043.324} C_VEL
LIN {X 0,Y 460.477,Z 364.127,A -85,B 0,C 180,E1 -8046.528,E2 -8046.528} C_VEL
LIN {X 0,Y 460.581,Z 364.114,A -85,B 0,C 180,E1 -8049.856,E2 -8049.856} C_VEL
LIN {X 0,Y 460.509,Z 364.117,A -85,B 0,C 180,E1 -8052.9,E2 -8052.9} C_VEL
LIN {X 0,Y 460.519,Z 364.122,A -85,B 0,C 180,E1 -8055.828,E2 -8055.828} C_VEL
LIN {X 0,Y 460.538,Z 364.115,A -85,B 0,C 180,E1 -8058.989,E2 -8058.989} C_VEL
LIN {X 0,Y 460.541,Z 364.115,A -85,B 0,C 180,E1 -8061.268,E2 -8061.268} C_VEL
LIN {X 0,Y 460.507,Z 364.119,A -85,B 0,C 180,E1 -8064.554,E2 -8064.554} C_VEL
LIN {X 0,Y 460.526,Z 364.121,A -85,B 0,C 180,E1 -8067.715,E2 -8067.715} C_VEL
LIN {X 0,Y 460.54,Z 364.112,A -85,B 0,C 180,E1 -8070.769,E2 -8070.769} C_VEL
LIN {X 0,Y 460.56,Z 364.113,A -85,B 0,C 180,E1 -8073.735,E2 -8073.735} C_VEL
LIN {X 0,Y 460.538,Z 364.114,A -85,B 0,C 180,E1 -8076.624,E2 -8076.624} C_VEL
LIN {X 0,Y 460.543,Z 364.116,A -85,B 0,C 180,E1 -8079.452,E2 -8079.452} C_VEL
LIN {X 0,Y 460.55,Z 364.109,A -85,B 0,C 180,E1 -8082.23,E2 -8082.23} C_VEL
LIN {X 0,Y 460.562,Z 364.113,A -85,B 0,C 180,E1 -8084.965,E2 -8084.965} C_VEL
LIN {X 0,Y 460.604,Z 364.104,A -85,B 0,C 180,E1 -8088.559,E2 -8088.559} C_VEL
LIN {X 0,Y 460.686,Z 364.091,A -85,B 0,C 180,E1 -8092.109,E2 -8092.109} C_VEL
LIN {X 0,Y 460.69,Z 364.096,A -85,B 0,C 180,E1 -8094.748,E2 -8094.748} C_VEL
LIN {X 0,Y 460.817,Z 364.081,A -85,B 0,C 180,E1 -8097.378,E2 -8097.378} C_VEL
LIN {X 0,Y 460.844,Z 364.077,A -85,B 0,C 180,E1 -8100,E2 -8100} C_VEL
LIN {X 0,Y 460.818,Z 364.075,A -85,B 0,C 180,E1 -8102.623,E2 -8102.623} C_VEL
LIN {X 0,Y 460.704,Z 364.092,A -85,B 0,C 180,E1 -8106.13,E2 -8106.13} C_VEL
LIN {X 0,Y 460.621,Z 364.104,A -85,B 0,C 180,E1 -8108.777,E2 -8108.777} C_VEL
LIN {X 0,Y 460.605,Z 364.102,A -85,B 0,C 180,E1 -8112.445,E2 -8112.445} C_VEL
LIN {X 0,Y 460.592,Z 364.104,A -85,B 0,C 180,E1 -8115.998,E2 -8115.998} C_VEL
LIN {X 0,Y 460.564,Z 364.117,A -85,B 0,C 180,E1 -8118.903,E2 -8118.903} C_VEL
LIN {X 0,Y 460.554,Z 364.116,A -85,B 0,C 180,E1 -8121.484,E2 -8121.484} C_VEL
LIN {X 0,Y 460.538,Z 364.112,A -85,B 0,C 180,E1 -8124.333,E2 -8124.333} C_VEL
LIN {X 0,Y 460.578,Z 364.113,A -85,B 0,C 180,E1 -8127.244,E2 -8127.244} C_VEL
LIN {X 0,Y 460.505,Z 364.119,A -85,B 0,C 180,E1 -8130.241,E2 -8130.241} C_VEL
LIN {X 0,Y 460.524,Z 364.113,A -85,B 0,C 180,E1 -8133.326,E2 -8133.326} C_VEL
LIN {X 0,Y 460.475,Z 364.127,A -85,B 0,C 180,E1 -8136.53,E2 -8136.53} C_VEL
LIN {X 0,Y 460.571,Z 364.11,A -85,B 0,C 180,E1 -8139.859,E2 -8139.859} C_VEL
LIN {X 0,Y 460.54,Z 364.118,A -85,B 0,C 180,E1 -8142.905,E2 -8142.905} C_VEL
LIN {X 0,Y 460.517,Z 364.118,A -85,B 0,C 180,E1 -8145.83,E2 -8145.83} C_VEL
LIN {X 0,Y 460.533,Z 364.122,A -85,B 0,C 180,E1 -8148.99,E2 -8148.99} C_VEL
LIN {X 0,Y 460.526,Z 364.124,A -85,B 0,C 180,E1 -8151.268,E2 -8151.268} C_VEL
LIN {X 0,Y 460.52,Z 364.15,A -85,B 0,C 180,E1 -8153.203,E2 -8153.203} C_VEL
LIN {X 0,Y 461.89,Z 371.47,A -85,B 0,C 180,E1 -8155.007,E2 -8155.007} C_VEL
LIN {X 0,Y 461.674,Z 378.926,A -85,B 0,C 180,E1 -8156.718,E2 -8156.718} C_VEL
LIN {X 0,Y 464.81,Z 393.32,A -85,B 0,C 180,E1 -8157.083,E2 -8157.083} C_VEL
LIN {X 0,Y 463.937,Z 485.701,A -85,B 0,C 180,E1 -8158.556,E2 -8158.556} C_VEL
LIN {X 0,Y 463.583,Z 498.809,A -85,B 0,C 180,E1 -8158.942,E2 -8158.942} C_VEL
LIN {X 0,Y 463.236,Z 511.913,A -85,B 0,C 180,E1 -8159.523,E2 -8159.523} C_VEL
LIN {X 0,Y 462.811,Z 522.82,A -85,B 0,C 180,E1 -8160.178,E2 -8160.178} C_VEL
LIN {X 0,Y 462.321,Z 533.809,A -85,B 0,C 180,E1 -8161.018,E2 -8161.018} C_VEL
LIN {X 0,Y 462.133,Z 537.212,A -85,B 0,C 180,E1 -8161.316,E2 -8161.316} C_VEL
LIN {X 0,Y 461.224,Z 541.968,A -85,B 0,C 180,E1 -8161.752,E2 -8161.752} C_VEL
LIN {X 0,Y 457.991,Z 549.417,A -85,B 0,C 180,E1 -8162.471,E2 -8162.471} C_VEL
LIN {X 0,Y 454.799,Z 556.276,A -85,B 0,C 180,E1 -8163.265,E2 -8163.265} C_VEL
LIN {X 0,Y 453.948,Z 560.112,A -85,B 0,C 180,E1 -8163.81,E2 -8163.81} C_VEL
LIN {X 0,Y 453.509,Z 567.237,A -85,B 0,C 180,E1 -8165.021,E2 -8165.021} C_VEL
LIN {X 0,Y 453.212,Z 573.022,A -85,B 0,C 180,E1 -8166.223,E2 -8166.223} C_VEL
LIN {X 0,Y 452.912,Z 578.57,A -85,B 0,C 180,E1 -8167.656,E2 -8167.656} C_VEL
LIN {X 0,Y 452.719,Z 582.778,A -85,B 0,C 180,E1 -8169.081,E2 -8169.081} C_VEL
LIN {X 0,Y 452.601,Z 584.896,A -85,B 0,C 180,E1 -8170.025,E2 -8170.025} C_VEL
LIN {X 0,Y 452.491,Z 587.092,A -85,B 0,C 180,E1 -8171.343,E2 -8171.343} C_VEL
LIN {X 0,Y 452.377,Z 588.496,A -85,B 0,C 180,E1 -8172.832,E2 -8172.832} C_VEL
LIN {X 0,Y 452.427,Z 588.782,A -85,B 0,C 180,E1 -8174.39,E2 -8174.39} C_VEL
LIN {X 0,Y 452.429,Z 588.181,A -85,B 0,C 180,E1 -8175.609,E2 -8175.609} C_VEL
LIN {X 0,Y 452.453,Z 587.222,A -85,B 0,C 180,E1 -8176.527,E2 -8176.527} C_VEL
LIN {X 0,Y 452.609,Z 584.729,A -85,B 0,C 180,E1 -8178.03,E2 -8178.03} C_VEL
LIN {X 0,Y 452.774,Z 580.476,A -85,B 0,C 180,E1 -8179.718,E2 -8179.718} C_VEL
LIN {X 0,Y 453.003,Z 575.782,A -85,B 0,C 180,E1 -8181.075,E2 -8181.075} C_VEL
LIN {X 0,Y 453.305,Z 569.618,A -85,B 0,C 180,E1 -8182.472,E2 -8182.472} C_VEL
LIN {X 0,Y 453.625,Z 562.464,A -85,B 0,C 180,E1 -8183.774,E2 -8183.774} C_VEL
LIN {X 0,Y 454.073,Z 554.93,A -85,B 0,C 180,E1 -8184.894,E2 -8184.894} C_VEL
LIN {X 0,Y 454.528,Z 545.844,A -85,B 0,C 180,E1 -8186.01,E2 -8186.01} C_VEL
LIN {X 0,Y 455.103,Z 535.732,A -85,B 0,C 180,E1 -8187.013,E2 -8187.013} C_VEL
LIN {X 0,Y 455.609,Z 524.552,A -85,B 0,C 180,E1 -8187.901,E2 -8187.901} C_VEL
LIN {X 0,Y 456.087,Z 513.945,A -85,B 0,C 180,E1 -8188.565,E2 -8188.565} C_VEL
LIN {X 0,Y 456.453,Z 501.085,A -85,B 0,C 180,E1 -8189.178,E2 -8189.178} C_VEL
LIN {X 0,Y 456.731,Z 488.955,A -85,B 0,C 180,E1 -8189.573,E2 -8189.573} C_VEL
LIN {X 0,Y 456.988,Z 470.636,A -85,B 0,C 180,E1 -8189.913,E2 -8189.913} C_VEL
LIN {X 0,Y 457.626,Z 393.884,A -85,B 0,C 180,E1 -8191.126,E2 -8191.126} C_VEL
LIN {X 0,Y 454.573,Z 378.853,A -85,B 0,C 180,E1 -8191.495,E2 -8191.495} C_VEL
LIN {X 0,Y 454.817,Z 371.783,A -85,B 0,C 180,E1 -8193.1,E2 -8193.1} C_VEL
LIN {X 0,Y 453.558,Z 364.99,A -85,B 0,C 180,E1 -8194.777,E2 -8194.777} C_VEL
LIN {X 0,Y 453.64,Z 364.981,A -85,B 0,C 180,E1 -8197.464,E2 -8197.464} C_VEL
LIN {X 0,Y 453.537,Z 364.987,A -85,B 0,C 180,E1 -8200.716,E2 -8200.716} C_VEL
LIN {X 0,Y 453.515,Z 364.996,A -85,B 0,C 180,E1 -8203.441,E2 -8203.441} C_VEL
LIN {X 0,Y 453.549,Z 364.984,A -85,B 0,C 180,E1 -8206.195,E2 -8206.195} C_VEL
LIN {X 0,Y 453.525,Z 364.992,A -85,B 0,C 180,E1 -8209.04,E2 -8209.04} C_VEL
LIN {X 0,Y 453.481,Z 364.995,A -85,B 0,C 180,E1 -8211.835,E2 -8211.835} C_VEL
LIN {X 0,Y 453.517,Z 364.99,A -85,B 0,C 180,E1 -8214.734,E2 -8214.734} C_VEL
LIN {X 0,Y 453.534,Z 364.987,A -85,B 0,C 180,E1 -8217.959,E2 -8217.959} C_VEL
LIN {X 0,Y 453.488,Z 364.996,A -85,B 0,C 180,E1 -8221.528,E2 -8221.528} C_VEL
LIN {X 0,Y 453.49,Z 364.995,A -85,B 0,C 180,E1 -8224.777,E2 -8224.777} C_VEL
LIN {X 0,Y 453.476,Z 364.994,A -85,B 0,C 180,E1 -8228.309,E2 -8228.309} C_VEL
LIN {X 0,Y 453.493,Z 364.994,A -85,B 0,C 180,E1 -8230.608,E2 -8230.608} C_VEL
LIN {X 0,Y 453.455,Z 365.001,A -85,B 0,C 180,E1 -8233.243,E2 -8233.243} C_VEL
LIN {X 0,Y 453.474,Z 364.994,A -85,B 0,C 180,E1 -8235.779,E2 -8235.779} C_VEL
LIN {X 0,Y 453.491,Z 364.994,A -85,B 0,C 180,E1 -8239.39,E2 -8239.39} C_VEL
LIN {X 0,Y 453.47,Z 364.995,A -85,B 0,C 180,E1 -8242.222,E2 -8242.222} C_VEL
LIN {X 0,Y 453.484,Z 364.996,A -85,B 0,C 180,E1 -8245.221,E2 -8245.221} C_VEL
LIN {X 0,Y 453.461,Z 364.998,A -85,B 0,C 180,E1 -8248.474,E2 -8248.474} C_VEL
LIN {X 0,Y 453.531,Z 364.987,A -85,B 0,C 180,E1 -8252.038,E2 -8252.038} C_VEL
LIN {X 0,Y 453.508,Z 364.992,A -85,B 0,C 180,E1 -8255.265,E2 -8255.265} C_VEL
LIN {X 0,Y 453.473,Z 364.997,A -85,B 0,C 180,E1 -8258.414,E2 -8258.414} C_VEL
LIN {X 0,Y 453.515,Z 364.993,A -85,B 0,C 180,E1 -8261.008,E2 -8261.008} C_VEL
LIN {X 0,Y 453.56,Z 364.983,A -85,B 0,C 180,E1 -8263.879,E2 -8263.879} C_VEL
LIN {X 0,Y 453.555,Z 364.984,A -85,B 0,C 180,E1 -8267.471,E2 -8267.471} C_VEL
LIN {X 0,Y 453.585,Z 364.982,A -85,B 0,C 180,E1 -8271.086,E2 -8271.086} C_VEL
LIN {X 0,Y 453.671,Z 364.969,A -85,B 0,C 180,E1 -8273.774,E2 -8273.774} C_VEL
LIN {X 0,Y 453.757,Z 364.959,A -85,B 0,C 180,E1 -8277.337,E2 -8277.337} C_VEL
LIN {X 0,Y 453.814,Z 364.953,A -85,B 0,C 180,E1 -8280,E2 -8280} C_VEL
LIN {X 0,Y 453.757,Z 364.964,A -85,B 0,C 180,E1 -8282.663,E2 -8282.663} C_VEL
LIN {X 0,Y 453.668,Z 364.974,A -85,B 0,C 180,E1 -8286.225,E2 -8286.225} C_VEL
LIN {X 0,Y 453.584,Z 364.982,A -85,B 0,C 180,E1 -8288.913,E2 -8288.913} C_VEL
LIN {X 0,Y 453.554,Z 364.99,A -85,B 0,C 180,E1 -8292.529,E2 -8292.529} C_VEL
LIN {X 0,Y 453.548,Z 364.991,A -85,B 0,C 180,E1 -8296.196,E2 -8296.196} C_VEL
LIN {X 0,Y 453.512,Z 364.99,A -85,B 0,C 180,E1 -8299.041,E2 -8299.041} C_VEL
LIN {X 0,Y 453.468,Z 364.997,A -85,B 0,C 180,E1 -8301.836,E2 -8301.836} C_VEL
LIN {X 0,Y 453.506,Z 364.992,A -85,B 0,C 180,E1 -8304.735,E2 -8304.735} C_VEL
LIN {X 0,Y 453.531,Z 364.991,A -85,B 0,C 180,E1 -8307.962,E2 -8307.962} C_VEL
LIN {X 0,Y 453.476,Z 364.995,A -85,B 0,C 180,E1 -8310.759,E2 -8310.759} C_VEL
LIN {X 0,Y 453.472,Z 364.999,A -85,B 0,C 180,E1 -8313.913,E2 -8313.913} C_VEL
LIN {X 0,Y 453.466,Z 364.995,A -85,B 0,C 180,E1 -8317.188,E2 -8317.188} C_VEL
LIN {X 0,Y 453.528,Z 364.988,A -85,B 0,C 180,E1 -8319.446,E2 -8319.446} C_VEL
LIN {X 0,Y 453.487,Z 364.992,A -85,B 0,C 180,E1 -8322.992,E2 -8322.992} C_VEL
LIN {X 0,Y 453.462,Z 365,A -85,B 0,C 180,E1 -8325.78,E2 -8325.78} C_VEL
LIN {X 0,Y 453.513,Z 364.99,A -85,B 0,C 180,E1 -8329.406,E2 -8329.406} C_VEL
LIN {X 0,Y 453.476,Z 364.998,A -85,B 0,C 180,E1 -8332.223,E2 -8332.223} C_VEL
LIN {X 0,Y 453.487,Z 364.993,A -85,B 0,C 180,E1 -8335.223,E2 -8335.223} C_VEL
LIN {X 0,Y 453.468,Z 364.996,A -85,B 0,C 180,E1 -8338.475,E2 -8338.475} C_VEL
LIN {X 0,Y 453.515,Z 364.996,A -85,B 0,C 180,E1 -8341.289,E2 -8341.289} C_VEL
LIN {X 0,Y 453.619,Z 365.172,A -85,B 0,C 180,E1 -8343.053,E2 -8343.053} C_VEL
LIN {X 0,Y 456.157,Z 378.244,A -85,B 0,C 180,E1 -8345.545,E2 -8345.545} C_VEL
LIN {X 0,Y 455.512,Z 392.266,A -85,B 0,C 180,E1 -8348.01,E2 -8348.01} C_VEL
LIN {X 0,Y 454.634,Z 411.172,A -85,B 0,C 180,E1 -8351.291,E2 -8351.291} C_VEL
LIN {X 0,Y 454.322,Z 418.46,A -85,B 0,C 180,E1 -8352.52,E2 -8352.52} C_VEL
LIN {X 0,Y 457.442,Z 439.479,A -85,B 0,C 180,E1 -8352.969,E2 -8352.969} C_VEL
LIN {X 0,Y 456.708,Z 527.275,A -85,B 0,C 180,E1 -8354.378,E2 -8354.378} C_VEL
LIN {X 0,Y 456.285,Z 540.428,A -85,B 0,C 180,E1 -8354.764,E2 -8354.764} C_VEL
LIN {X 0,Y 455.793,Z 553.123,A -85,B 0,C 180,E1 -8355.318,E2 -8355.318} C_VEL
LIN {X 0,Y 455.205,Z 565.2,A -85,B 0,C 180,E1 -8356.041,E2 -8356.041} C_VEL
LIN {X 0,Y 454.572,Z 577.432,A -85,B 0,C 180,E1 -8356.992,E2 -8356.992} C_VEL
LIN {X 0,Y 454.173,Z 587.158,A -85,B 0,C 180,E1 -8357.942,E2 -8357.942} C_VEL
LIN {X 0,Y 453.65,Z 596.491,A -85,B 0,C 180,E1 -8359.06,E2 -8359.06} C_VEL
LIN {X 0,Y 453.167,Z 605.543,A -85,B 0,C 180,E1 -8360.403,E2 -8360.403} C_VEL
LIN {X 0,Y 452.863,Z 612.838,A -85,B 0,C 180,E1 -8361.747,E2 -8361.747} C_VEL
LIN {X 0,Y 452.694,Z 617.764,A -85,B 0,C 180,E1 -8362.866,E2 -8362.866} C_VEL
LIN {X 0,Y 452.557,Z 622.55,A -85,B 0,C 180,E1 -8364.207,E2 -8364.207} C_VEL
LIN {X 0,Y 452.494,Z 626.209,A -85,B 0,C 180,E1 -8365.546,E2 -8365.546} C_VEL
LIN {X 0,Y 452.494,Z 628.1,A -85,B 0,C 180,E1 -8366.438,E2 -8366.438} C_VEL
LIN {X 0,Y 452.523,Z 629.524,A -85,B 0,C 180,E1 -8367.33,E2 -8367.33} C_VEL
LIN {X 0,Y 452.488,Z 631.151,A -85,B 0,C 180,E1 -8369.11,E2 -8369.11} C_VEL
LIN {X 0,Y 452.465,Z 631.377,A -85,B 0,C 180,E1 -8370,E2 -8370} C_VEL
LIN {X 0,Y 452.488,Z 631.173,A -85,B 0,C 180,E1 -8370.89,E2 -8370.89} C_VEL
LIN {X 0,Y 452.523,Z 629.57,A -85,B 0,C 180,E1 -8372.67,E2 -8372.67} C_VEL
LIN {X 0,Y 452.492,Z 628.173,A -85,B 0,C 180,E1 -8373.562,E2 -8373.562} C_VEL
LIN {X 0,Y 452.551,Z 625.232,A -85,B 0,C 180,E1 -8374.9,E2 -8374.9} C_VEL
LIN {X 0,Y 452.61,Z 620.726,A -85,B 0,C 180,E1 -8376.396,E2 -8376.396} C_VEL
LIN {X 0,Y 452.802,Z 615.149,A -85,B 0,C 180,E1 -8377.805,E2 -8377.805} C_VEL
LIN {X 0,Y 453.057,Z 608.479,A -85,B 0,C 180,E1 -8379.149,E2 -8379.149} C_VEL
LIN {X 0,Y 453.46,Z 600.219,A -85,B 0,C 180,E1 -8380.492,E2 -8380.492} C_VEL
LIN {X 0,Y 453.961,Z 591.784,A -85,B 0,C 180,E1 -8381.61,E2 -8381.61} C_VEL
LIN {X 0,Y 454.466,Z 582.339,A -85,B 0,C 180,E1 -8382.639,E2 -8382.639} C_VEL
LIN {X 0,Y 455.029,Z 571.126,A -85,B 0,C 180,E1 -8383.623,E2 -8383.623} C_VEL
LIN {X 0,Y 455.641,Z 559.922,A -85,B 0,C 180,E1 -8384.401,E2 -8384.401} C_VEL
LIN {X 0,Y 456.246,Z 547.378,A -85,B 0,C 180,E1 -8385.066,E2 -8385.066} C_VEL
LIN {X 0,Y 456.732,Z 533.984,A -85,B 0,C 180,E1 -8385.564,E2 -8385.564} C_VEL
LIN {X 0,Y 457.039,Z 520.829,A -85,B 0,C 180,E1 -8385.868,E2 -8385.868} C_VEL
LIN {X 0,Y 457.685,Z 439.361,A -85,B 0,C 180,E1 -8387.167,E2 -8387.167} C_VEL
LIN {X 0,Y 454.42,Z 417.953,A -85,B 0,C 180,E1 -8387.659,E2 -8387.659} C_VEL
LIN {X 0,Y 455.266,Z 400.082,A -85,B 0,C 180,E1 -8390.796,E2 -8390.796} C_VEL
LIN {X 0,Y 456.239,Z 382.95,A -85,B 0,C 180,E1 -8393.85,E2 -8393.85} C_VEL
LIN {X 0,Y 456.279,Z 378.524,A -85,B 0,C 180,E1 -8394.664,E2 -8394.664} C_VEL
LIN {X 0,Y 454.058,Z 367.18,A -85,B 0,C 180,E1 -8396.919,E2 -8396.919} C_VEL
LIN {X 0,Y 453.575,Z 364.988,A -85,B 0,C 180,E1 -8397.386,E2 -8397.386} C_VEL
LIN {X 0,Y 453.482,Z 364.996,A -85,B 0,C 180,E1 -8400.758,E2 -8400.758} C_VEL
LIN {X 0,Y 453.477,Z 364.998,A -85,B 0,C 180,E1 -8403.912,E2 -8403.912} C_VEL
LIN {X 0,Y 453.47,Z 364.998,A -85,B 0,C 180,E1 -8407.187,E2 -8407.187} C_VEL
LIN {X 0,Y 453.534,Z 364.988,A -85,B 0,C 180,E1 -8409.444,E2 -8409.444} C_VEL
LIN {X 0,Y 453.459,Z 364.995,A -85,B 0,C 180,E1 -8412.994,E2 -8412.994} C_VEL
LIN {X 0,Y 453.472,Z 364.999,A -85,B 0,C 180,E1 -8415.78,E2 -8415.78} C_VEL
LIN {X 0,Y 453.491,Z 364.997,A -85,B 0,C 180,E1 -8418.211,E2 -8418.211} C_VEL
LIN {X 0,Y 453.527,Z 364.988,A -85,B 0,C 180,E1 -8420.787,E2 -8420.787} C_VEL
LIN {X 0,Y 453.451,Z 365.003,A -85,B 0,C 180,E1 -8423.917,E2 -8423.917} C_VEL
LIN {X 0,Y 453.476,Z 364.993,A -85,B 0,C 180,E1 -8427.151,E2 -8427.151} C_VEL
LIN {X 0,Y 453.507,Z 364.99,A -85,B 0,C 180,E1 -8430.271,E2 -8430.271} C_VEL
LIN {X 0,Y 453.506,Z 364.993,A -85,B 0,C 180,E1 -8433.294,E2 -8433.294} C_VEL
LIN {X 0,Y 453.495,Z 364.993,A -85,B 0,C 180,E1 -8436.238,E2 -8436.238} C_VEL
LIN {X 0,Y 453.474,Z 364.993,A -85,B 0,C 180,E1 -8439.117,E2 -8439.117} C_VEL
LIN {X 0,Y 453.503,Z 364.99,A -85,B 0,C 180,E1 -8441.944,E2 -8441.944} C_VEL
LIN {X 0,Y 453.542,Z 364.986,A -85,B 0,C 180,E1 -8444.727,E2 -8444.727} C_VEL
LIN {X 0,Y 453.552,Z 364.982,A -85,B 0,C 180,E1 -8448.379,E2 -8448.379} C_VEL
LIN {X 0,Y 453.643,Z 364.969,A -85,B 0,C 180,E1 -8451.985,E2 -8451.985} C_VEL
LIN {X 0,Y 453.663,Z 364.971,A -85,B 0,C 180,E1 -8454.667,E2 -8454.667} C_VEL
LIN {X 0,Y 453.758,Z 364.96,A -85,B 0,C 180,E1 -8457.337,E2 -8457.337} C_VEL
LIN {X 0,Y 453.815,Z 364.953,A -85,B 0,C 180,E1 -8460,E2 -8460} C_VEL
LIN {X 0,Y 453.758,Z 364.955,A -85,B 0,C 180,E1 -8462.663,E2 -8462.663} C_VEL
LIN {X 0,Y 453.671,Z 364.968,A -85,B 0,C 180,E1 -8466.226,E2 -8466.226} C_VEL
LIN {X 0,Y 453.585,Z 364.982,A -85,B 0,C 180,E1 -8468.914,E2 -8468.914} C_VEL
LIN {X 0,Y 453.555,Z 364.981,A -85,B 0,C 180,E1 -8472.529,E2 -8472.529} C_VEL
LIN {X 0,Y 453.537,Z 364.983,A -85,B 0,C 180,E1 -8476.197,E2 -8476.197} C_VEL
LIN {X 0,Y 453.513,Z 364.995,A -85,B 0,C 180,E1 -8479.042,E2 -8479.042} C_VEL
LIN {X 0,Y 453.491,Z 364.993,A -85,B 0,C 180,E1 -8481.836,E2 -8481.836} C_VEL
LIN {X 0,Y 453.509,Z 364.991,A -85,B 0,C 180,E1 -8484.735,E2 -8484.735} C_VEL
LIN {X 0,Y 453.532,Z 364.987,A -85,B 0,C 180,E1 -8487.962,E2 -8487.962} C_VEL
LIN {X 0,Y 453.461,Z 364.999,A -85,B 0,C 180,E1 -8491.526,E2 -8491.526} C_VEL
LIN {X 0,Y 453.485,Z 364.99,A -85,B 0,C 180,E1 -8494.779,E2 -8494.779} C_VEL
LIN {X 0,Y 453.479,Z 364.996,A -85,B 0,C 180,E1 -8498.311,E2 -8498.311} C_VEL
LIN {X 0,Y 453.513,Z 364.995,A -85,B 0,C 180,E1 -8500.607,E2 -8500.607} C_VEL
LIN {X 0,Y 453.48,Z 364.998,A -85,B 0,C 180,E1 -8503.249,E2 -8503.249} C_VEL
LIN {X 0,Y 453.471,Z 364.996,A -85,B 0,C 180,E1 -8505.781,E2 -8505.781} C_VEL
LIN {X 0,Y 453.48,Z 364.997,A -85,B 0,C 180,E1 -8508.211,E2 -8508.211} C_VEL
LIN {X 0,Y 453.515,Z 364.996,A -85,B 0,C 180,E1 -8510.791,E2 -8510.791} C_VEL
LIN {X 0,Y 453.484,Z 365.065,A -85,B 0,C 180,E1 -8512.977,E2 -8512.977} C_VEL
LIN {X 0,Y 454.969,Z 372.984,A -85,B 0,C 180,E1 -8514.956,E2 -8514.956} C_VEL
LIN {X 0,Y 454.791,Z 379.167,A -85,B 0,C 180,E1 -8516.397,E2 -8516.397} C_VEL
LIN {X 0,Y 458.084,Z 394.248,A -85,B 0,C 180,E1 -8516.813,E2 -8516.813} C_VEL
LIN {X 0,Y 457.179,Z 485.408,A -85,B 0,C 180,E1 -8518.284,E2 -8518.284} C_VEL
LIN {X 0,Y 456.791,Z 499.005,A -85,B 0,C 180,E1 -8518.686,E2 -8518.686} C_VEL
LIN {X 0,Y 456.448,Z 512.044,A -85,B 0,C 180,E1 -8519.271,E2 -8519.271} C_VEL
LIN {X 0,Y 455.937,Z 523.688,A -85,B 0,C 180,E1 -8519.982,E2 -8519.982} C_VEL
LIN {X 0,Y 455.381,Z 535.479,A -85,B 0,C 180,E1 -8520.913,E2 -8520.913} C_VEL
LIN {X 0,Y 454.856,Z 544.823,A -85,B 0,C 180,E1 -8521.831,E2 -8521.831} C_VEL
LIN {X 0,Y 454.321,Z 553.38,A -85,B 0,C 180,E1 -8522.849,E2 -8522.849} C_VEL
LIN {X 0,Y 453.948,Z 560.112,A -85,B 0,C 180,E1 -8523.81,E2 -8523.81} C_VEL
LIN {X 0,Y 453.104,Z 563.811,A -85,B 0,C 180,E1 -8524.383,E2 -8524.383} C_VEL
LIN {X 0,Y 449.936,Z 569.466,A -85,B 0,C 180,E1 -8525.338,E2 -8525.338} C_VEL
LIN {X 0,Y 446.774,Z 574.463,A -85,B 0,C 180,E1 -8526.358,E2 -8526.358} C_VEL
LIN {X 0,Y 445.955,Z 577.114,A -85,B 0,C 180,E1 -8527.029,E2 -8527.029} C_VEL
LIN {X 0,Y 445.726,Z 581.776,A -85,B 0,C 180,E1 -8528.481,E2 -8528.481} C_VEL
LIN {X 0,Y 445.563,Z 584.758,A -85,B 0,C 180,E1 -8529.696,E2 -8529.696} C_VEL
LIN {X 0,Y 445.424,Z 587.344,A -85,B 0,C 180,E1 -8531.21,E2 -8531.21} C_VEL
LIN {X 0,Y 445.298,Z 588.705,A -85,B 0,C 180,E1 -8532.551,E2 -8532.551} C_VEL
LIN {X 0,Y 445.33,Z 589.13,A -85,B 0,C 180,E1 -8534.298,E2 -8534.298} C_VEL
LIN {X 0,Y 445.34,Z 588.7,A -85,B 0,C 180,E1 -8535.375,E2 -8535.375} C_VEL
LIN {X 0,Y 445.371,Z 587.847,A -85,B 0,C 180,E1 -8536.308,E2 -8536.308} C_VEL
LIN {X 0,Y 445.534,Z 585.272,A -85,B 0,C 180,E1 -8537.964,E2 -8537.964} C_VEL
LIN {X 0,Y 445.684,Z 581.478,A -85,B 0,C 180,E1 -8539.552,E2 -8539.552} C_VEL
LIN {X 0,Y 445.897,Z 576.992,A -85,B 0,C 180,E1 -8540.932,E2 -8540.932} C_VEL
LIN {X 0,Y 446.27,Z 570.185,A -85,B 0,C 180,E1 -8542.535,E2 -8542.535} C_VEL
LIN {X 0,Y 446.62,Z 562.808,A -85,B 0,C 180,E1 -8543.903,E2 -8543.903} C_VEL
LIN {X 0,Y 447.077,Z 555.28,A -85,B 0,C 180,E1 -8545.04,E2 -8545.04} C_VEL
LIN {X 0,Y 447.555,Z 546.198,A -85,B 0,C 180,E1 -8546.173,E2 -8546.173} C_VEL
LIN {X 0,Y 448.155,Z 536.093,A -85,B 0,C 180,E1 -8547.191,E2 -8547.191} C_VEL
LIN {X 0,Y 448.698,Z 524.913,A -85,B 0,C 180,E1 -8548.093,E2 -8548.093} C_VEL
LIN {X 0,Y 449.204,Z 514.309,A -85,B 0,C 180,E1 -8548.767,E2 -8548.767} C_VEL
LIN {X 0,Y 449.559,Z 502.396,A -85,B 0,C 180,E1 -8549.351,E2 -8549.351} C_VEL
LIN {X 0,Y 449.851,Z 490.065,A -85,B 0,C 180,E1 -8549.773,E2 -8549.773} C_VEL
LIN {X 0,Y 450.119,Z 474.29,A -85,B 0,C 180,E1 -8550.084,E2 -8550.084} C_VEL
LIN {X 0,Y 450.764,Z 394.539,A -85,B 0,C 180,E1 -8551.363,E2 -8551.363} C_VEL
LIN {X 0,Y 447.628,Z 379.089,A -85,B 0,C 180,E1 -8551.761,E2 -8551.761} C_VEL
LIN {X 0,Y 447.842,Z 373.067,A -85,B 0,C 180,E1 -8553.149,E2 -8553.149} C_VEL
LIN {X 0,Y 446.534,Z 365.865,A -85,B 0,C 180,E1 -8554.909,E2 -8554.909} C_VEL
LIN {X 0,Y 446.593,Z 365.859,A -85,B 0,C 180,E1 -8557.504,E2 -8557.504} C_VEL
LIN {X 0,Y 446.489,Z 365.866,A -85,B 0,C 180,E1 -8560.888,E2 -8560.888} C_VEL
LIN {X 0,Y 446.473,Z 365.87,A -85,B 0,C 180,E1 -8563.657,E2 -8563.657} C_VEL
LIN {X 0,Y 446.495,Z 365.863,A -85,B 0,C 180,E1 -8566.458,E2 -8566.458} C_VEL
LIN {X 0,Y 446.473,Z 365.874,A -85,B 0,C 180,E1 -8569.303,E2 -8569.303} C_VEL
LIN {X 0,Y 446.422,Z 365.872,A -85,B 0,C 180,E1 -8572.199,E2 -8572.199} C_VEL
LIN {X 0,Y 446.462,Z 365.874,A -85,B 0,C 180,E1 -8575.151,E2 -8575.151} C_VEL
LIN {X 0,Y 446.487,Z 365.864,A -85,B 0,C 180,E1 -8578.178,E2 -8578.178} C_VEL
LIN {X 0,Y 446.44,Z 365.871,A -85,B 0,C 180,E1 -8581.778,E2 -8581.778} C_VEL
LIN {X 0,Y 446.432,Z 365.878,A -85,B 0,C 180,E1 -8585.053,E2 -8585.053} C_VEL
LIN {X 0,Y 446.433,Z 365.871,A -85,B 0,C 180,E1 -8588.081,E2 -8588.081} C_VEL
LIN {X 0,Y 446.426,Z 365.878,A -85,B 0,C 180,E1 -8590.917,E2 -8590.917} C_VEL
LIN {X 0,Y 446.4,Z 365.875,A -85,B 0,C 180,E1 -8593.845,E2 -8593.845} C_VEL
LIN {X 0,Y 446.421,Z 365.874,A -85,B 0,C 180,E1 -8596.399,E2 -8596.399} C_VEL
LIN {X 0,Y 446.448,Z 365.869,A -85,B 0,C 180,E1 -8599.802,E2 -8599.802} C_VEL
LIN {X 0,Y 446.426,Z 365.872,A -85,B 0,C 180,E1 -8602.122,E2 -8602.122} C_VEL
LIN {X 0,Y 446.426,Z 365.873,A -85,B 0,C 180,E1 -8605.476,E2 -8605.476} C_VEL
LIN {X 0,Y 446.411,Z 365.879,A -85,B 0,C 180,E1 -8608.699,E2 -8608.699} C_VEL
LIN {X 0,Y 446.479,Z 365.865,A -85,B 0,C 180,E1 -8611.82,E2 -8611.82} C_VEL
LIN {X 0,Y 446.452,Z 365.876,A -85,B 0,C 180,E1 -8614.847,E2 -8614.847} C_VEL
LIN {X 0,Y 446.441,Z 365.872,A -85,B 0,C 180,E1 -8618.244,E2 -8618.244} C_VEL
LIN {X 0,Y 446.45,Z 365.869,A -85,B 0,C 180,E1 -8621.649,E2 -8621.649} C_VEL
LIN {X 0,Y 446.5,Z 365.868,A -85,B 0,C 180,E1 -8624.479,E2 -8624.479} C_VEL
LIN {X 0,Y 446.507,Z 365.862,A -85,B 0,C 180,E1 -8627.383,E2 -8627.383} C_VEL
LIN {X 0,Y 446.53,Z 365.863,A -85,B 0,C 180,E1 -8630.944,E2 -8630.944} C_VEL
LIN {X 0,Y 446.64,Z 365.845,A -85,B 0,C 180,E1 -8633.676,E2 -8633.676} C_VEL
LIN {X 0,Y 446.701,Z 365.838,A -85,B 0,C 180,E1 -8637.294,E2 -8637.294} C_VEL
LIN {X 0,Y 446.784,Z 365.829,A -85,B 0,C 180,E1 -8640,E2 -8640} C_VEL
LIN {X 0,Y 446.701,Z 365.843,A -85,B 0,C 180,E1 -8642.705,E2 -8642.705} C_VEL
LIN {X 0,Y 446.637,Z 365.852,A -85,B 0,C 180,E1 -8646.324,E2 -8646.324} C_VEL
LIN {X 0,Y 446.53,Z 365.86,A -85,B 0,C 180,E1 -8649.055,E2 -8649.055} C_VEL
LIN {X 0,Y 446.513,Z 365.864,A -85,B 0,C 180,E1 -8652.73,E2 -8652.73} C_VEL
LIN {X 0,Y 446.51,Z 365.868,A -85,B 0,C 180,E1 -8656.238,E2 -8656.238} C_VEL
LIN {X 0,Y 446.461,Z 365.867,A -85,B 0,C 180,E1 -8659.303,E2 -8659.303} C_VEL
LIN {X 0,Y 446.411,Z 365.881,A -85,B 0,C 180,E1 -8662.2,E2 -8662.2} C_VEL
LIN {X 0,Y 446.45,Z 365.869,A -85,B 0,C 180,E1 -8665.153,E2 -8665.153} C_VEL
LIN {X 0,Y 446.477,Z 365.873,A -85,B 0,C 180,E1 -8668.179,E2 -8668.179} C_VEL
LIN {X 0,Y 446.413,Z 365.873,A -85,B 0,C 180,E1 -8671.301,E2 -8671.301} C_VEL
LIN {X 0,Y 446.424,Z 365.875,A -85,B 0,C 180,E1 -8674.523,E2 -8674.523} C_VEL
LIN {X 0,Y 446.433,Z 365.879,A -85,B 0,C 180,E1 -8678.084,E2 -8678.084} C_VEL
LIN {X 0,Y 446.442,Z 365.87,A -85,B 0,C 180,E1 -8680.921,E2 -8680.921} C_VEL
LIN {X 0,Y 446.44,Z 365.875,A -85,B 0,C 180,E1 -8683.841,E2 -8683.841} C_VEL
LIN {X 0,Y 446.395,Z 365.879,A -85,B 0,C 180,E1 -8686.404,E2 -8686.404} C_VEL
LIN {X 0,Y 446.467,Z 365.872,A -85,B 0,C 180,E1 -8689.806,E2 -8689.806} C_VEL
LIN {X 0,Y 446.433,Z 365.876,A -85,B 0,C 180,E1 -8692.125,E2 -8692.125} C_VEL
LIN {X 0,Y 446.429,Z 365.874,A -85,B 0,C 180,E1 -8695.478,E2 -8695.478} C_VEL
LIN {X 0,Y 446.419,Z 365.873,A -85,B 0,C 180,E1 -8698.701,E2 -8698.701} C_VEL
LIN {X 0,Y 446.484,Z 365.875,A -85,B 0,C 180,E1 -8701.822,E2 -8701.822} C_VEL
LIN {X 0,Y 446.571,Z 366.028,A -85,B 0,C 180,E1 -8702.846,E2 -8702.846} C_VEL
LIN {X 0,Y 448.98,Z 378.237,A -85,B 0,C 180,E1 -8705.216,E2 -8705.216} C_VEL
LIN {X 0,Y 449.085,Z 382.475,A -85,B 0,C 180,E1 -8705.991,E2 -8705.991} C_VEL
LIN {X 0,Y 448.258,Z 398.623,A -85,B 0,C 180,E1 -8708.863,E2 -8708.863} C_VEL
LIN {X 0,Y 447.406,Z 416.198,A -85,B 0,C 180,E1 -8711.95,E2 -8711.95} C_VEL
LIN {X 0,Y 447.314,Z 417.971,A -85,B 0,C 180,E1 -8712.26,E2 -8712.26} C_VEL
LIN {X 0,Y 450.574,Z 441.433,A -85,B 0,C 180,E1 -8712.761,E2 -8712.761} C_VEL
LIN {X 0,Y 449.83,Z 527.169,A -85,B 0,C 180,E1 -8714.162,E2 -8714.162} C_VEL
LIN {X 0,Y 449.339,Z 541.008,A -85,B 0,C 180,E1 -8714.58,E2 -8714.58} C_VEL
LIN {X 0,Y 448.861,Z 553.441,A -85,B 0,C 180,E1 -8715.144,E2 -8715.144} C_VEL
LIN {X 0,Y 448.191,Z 566.14,A -85,B 0,C 180,E1 -8715.934,E2 -8715.934} C_VEL
LIN {X 0,Y 447.557,Z 577.944,A -85,B 0,C 180,E1 -8716.883,E2 -8716.883} C_VEL
LIN {X 0,Y 447.055,Z 588.622,A -85,B 0,C 180,E1 -8717.978,E2 -8717.978} C_VEL
LIN {X 0,Y 446.535,Z 597.641,A -85,B 0,C 180,E1 -8719.114,E2 -8719.114} C_VEL
LIN {X 0,Y 446.052,Z 606.447,A -85,B 0,C 180,E1 -8720.478,E2 -8720.478} C_VEL
LIN {X 0,Y 445.764,Z 613.472,A -85,B 0,C 180,E1 -8721.843,E2 -8721.843} C_VEL
LIN {X 0,Y 445.552,Z 619.257,A -85,B 0,C 180,E1 -8723.252,E2 -8723.252} C_VEL
LIN {X 0,Y 445.481,Z 624.759,A -85,B 0,C 180,E1 -8725.022,E2 -8725.022} C_VEL
LIN {X 0,Y 445.395,Z 627.737,A -85,B 0,C 180,E1 -8726.381,E2 -8726.381} C_VEL
LIN {X 0,Y 445.447,Z 629.173,A -85,B 0,C 180,E1 -8727.287,E2 -8727.287} C_VEL
LIN {X 0,Y 445.395,Z 630.809,A -85,B 0,C 180,E1 -8729.096,E2 -8729.096} C_VEL
LIN {X 0,Y 445.401,Z 631.043,A -85,B 0,C 180,E1 -8730,E2 -8730} C_VEL
LIN {X 0,Y 445.395,Z 630.846,A -85,B 0,C 180,E1 -8730.904,E2 -8730.904} C_VEL
LIN {X 0,Y 445.447,Z 629.254,A -85,B 0,C 180,E1 -8732.713,E2 -8732.713} C_VEL
LIN {X 0,Y 445.392,Z 627.863,A -85,B 0,C 180,E1 -8733.619,E2 -8733.619} C_VEL
LIN {X 0,Y 445.481,Z 624.935,A -85,B 0,C 180,E1 -8734.978,E2 -8734.978} C_VEL
LIN {X 0,Y 445.555,Z 619.554,A -85,B 0,C 180,E1 -8736.748,E2 -8736.748} C_VEL
LIN {X 0,Y 445.764,Z 613.882,A -85,B 0,C 180,E1 -8738.157,E2 -8738.157} C_VEL
LIN {X 0,Y 446.078,Z 607.011,A -85,B 0,C 180,E1 -8739.522,E2 -8739.522} C_VEL
LIN {X 0,Y 446.541,Z 598.462,A -85,B 0,C 180,E1 -8740.886,E2 -8740.886} C_VEL
LIN {X 0,Y 447.124,Z 589.69,A -85,B 0,C 180,E1 -8742.021,E2 -8742.021} C_VEL
LIN {X 0,Y 447.65,Z 579.629,A -85,B 0,C 180,E1 -8743.088,E2 -8743.088} C_VEL
LIN {X 0,Y 448.309,Z 568.168,A -85,B 0,C 180,E1 -8744.063,E2 -8744.063} C_VEL
LIN {X 0,Y 448.94,Z 556.137,A -85,B 0,C 180,E1 -8744.853,E2 -8744.853} C_VEL
LIN {X 0,Y 449.607,Z 543.619,A -85,B 0,C 180,E1 -8745.468,E2 -8745.468} C_VEL
LIN {X 0,Y 450.069,Z 530.546,A -85,B 0,C 180,E1 -8745.917,E2 -8745.917} C_VEL
LIN {X 0,Y 450.305,Z 514.85,A -85,B 0,C 180,E1 -8746.228,E2 -8746.228} C_VEL
LIN {X 0,Y 450.904,Z 439.47,A -85,B 0,C 180,E1 -8747.453,E2 -8747.453} C_VEL
LIN {X 0,Y 447.474,Z 417.515,A -85,B 0,C 180,E1 -8747.988,E2 -8747.988} C_VEL
LIN {X 0,Y 448.5,Z 398.616,A -85,B 0,C 180,E1 -8751.366,E2 -8751.366} C_VEL
LIN {X 0,Y 449.497,Z 381.708,A -85,B 0,C 180,E1 -8754.447,E2 -8754.447} C_VEL
LIN {X 0,Y 448.207,Z 373.666,A -85,B 0,C 180,E1 -8756.042,E2 -8756.042} C_VEL
LIN {X 0,Y 446.523,Z 365.866,A -85,B 0,C 180,E1 -8757.665,E2 -8757.665} C_VEL
LIN {X 0,Y 446.435,Z 365.88,A -85,B 0,C 180,E1 -8760.248,E2 -8760.248} C_VEL
LIN {X 0,Y 446.443,Z 365.871,A -85,B 0,C 180,E1 -8763.453,E2 -8763.453} C_VEL
LIN {X 0,Y 446.407,Z 365.878,A -85,B 0,C 180,E1 -8766.744,E2 -8766.744} C_VEL
LIN {X 0,Y 446.493,Z 365.865,A -85,B 0,C 180,E1 -8769.531,E2 -8769.531} C_VEL
LIN {X 0,Y 446.426,Z 365.872,A -85,B 0,C 180,E1 -8772.604,E2 -8772.604} C_VEL
LIN {X 0,Y 446.452,Z 365.87,A -85,B 0,C 180,E1 -8775.102,E2 -8775.102} C_VEL
LIN {X 0,Y 446.439,Z 365.872,A -85,B 0,C 180,E1 -8778.61,E2 -8778.61} C_VEL
LIN {X 0,Y 446.47,Z 365.867,A -85,B 0,C 180,E1 -8780.976,E2 -8780.976} C_VEL
LIN {X 0,Y 446.415,Z 365.876,A -85,B 0,C 180,E1 -8784.374,E2 -8784.374} C_VEL
LIN {X 0,Y 446.416,Z 365.877,A -85,B 0,C 180,E1 -8787.638,E2 -8787.638} C_VEL
LIN {X 0,Y 446.462,Z 365.866,A -85,B 0,C 180,E1 -8790.792,E2 -8790.792} C_VEL
LIN {X 0,Y 446.47,Z 365.868,A -85,B 0,C 180,E1 -8793.848,E2 -8793.848} C_VEL
LIN {X 0,Y 446.421,Z 365.873,A -85,B 0,C 180,E1 -8796.823,E2 -8796.823} C_VEL
LIN {X 0,Y 446.436,Z 365.878,A -85,B 0,C 180,E1 -8799.737,E2 -8799.737} C_VEL
LIN {X 0,Y 446.456,Z 365.864,A -85,B 0,C 180,E1 -8802.597,E2 -8802.597} C_VEL
LIN {X 0,Y 446.466,Z 365.874,A -85,B 0,C 180,E1 -8805.412,E2 -8805.412} C_VEL
LIN {X 0,Y 446.51,Z 365.86,A -85,B 0,C 180,E1 -8808.193,E2 -8808.193} C_VEL
LIN {X 0,Y 446.591,Z 365.848,A -85,B 0,C 180,E1 -8811.858,E2 -8811.858} C_VEL
LIN {X 0,Y 446.638,Z 365.846,A -85,B 0,C 180,E1 -8814.583,E2 -8814.583} C_VEL
LIN {X 0,Y 446.701,Z 365.838,A -85,B 0,C 180,E1 -8817.295,E2 -8817.295} C_VEL
LIN {X 0,Y 446.785,Z 365.829,A -85,B 0,C 180,E1 -8820,E2 -8820} C_VEL
LIN {X 0,Y 446.702,Z 365.834,A -85,B 0,C 180,E1 -8822.706,E2 -8822.706} C_VEL
LIN {X 0,Y 446.64,Z 365.844,A -85,B 0,C 180,E1 -8826.324,E2 -8826.324} C_VEL
LIN {X 0,Y 446.531,Z 365.863,A -85,B 0,C 180,E1 -8829.056,E2 -8829.056} C_VEL
LIN {X 0,Y 446.516,Z 365.859,A -85,B 0,C 180,E1 -8832.73,E2 -8832.73} C_VEL
LIN {X 0,Y 446.488,Z 365.861,A -85,B 0,C 180,E1 -8836.229,E2 -8836.229} C_VEL
LIN {X 0,Y 446.463,Z 365.87,A -85,B 0,C 180,E1 -8839.304,E2 -8839.304} C_VEL
LIN {X 0,Y 446.426,Z 365.873,A -85,B 0,C 180,E1 -8842.2,E2 -8842.2} C_VEL
LIN {X 0,Y 446.453,Z 365.876,A -85,B 0,C 180,E1 -8845.153,E2 -8845.153} C_VEL
LIN {X 0,Y 446.479,Z 365.866,A -85,B 0,C 180,E1 -8848.18,E2 -8848.18} C_VEL
LIN {X 0,Y 446.415,Z 365.876,A -85,B 0,C 180,E1 -8851.776,E2 -8851.776} C_VEL
LIN {X 0,Y 446.426,Z 365.868,A -85,B 0,C 180,E1 -8854.524,E2 -8854.524} C_VEL
LIN {X 0,Y 446.432,Z 365.872,A -85,B 0,C 180,E1 -8858.084,E2 -8858.084} C_VEL
LIN {X 0,Y 446.444,Z 365.875,A -85,B 0,C 180,E1 -8860.922,E2 -8860.922} C_VEL
LIN {X 0,Y 446.443,Z 365.873,A -85,B 0,C 180,E1 -8863.841,E2 -8863.841} C_VEL
LIN {X 0,Y 446.419,Z 365.879,A -85,B 0,C 180,E1 -8866.401,E2 -8866.401} C_VEL
LIN {X 0,Y 446.45,Z 365.873,A -85,B 0,C 180,E1 -8869.804,E2 -8869.804} C_VEL
LIN {X 0,Y 446.467,Z 365.975,A -85,B 0,C 180,E1 -8872.733,E2 -8872.733} C_VEL
LIN {X 0,Y 447.929,Z 373.576,A -85,B 0,C 180,E1 -8874.675,E2 -8874.675} C_VEL
LIN {X 0,Y 447.909,Z 379.461,A -85,B 0,C 180,E1 -8876.08,E2 -8876.08} C_VEL
LIN {X 0,Y 451.378,Z 395.162,A -85,B 0,C 180,E1 -8876.529,E2 -8876.529} C_VEL
LIN {X 0,Y 450.4,Z 486.175,A -85,B 0,C 180,E1 -8878.025,E2 -8878.025} C_VEL
LIN {X 0,Y 450.021,Z 499.763,A -85,B 0,C 180,E1 -8878.439,E2 -8878.439} C_VEL
LIN {X 0,Y 449.646,Z 512.379,A -85,B 0,C 180,E1 -8879.017,E2 -8879.017} C_VEL
LIN {X 0,Y 449.092,Z 524.403,A -85,B 0,C 180,E1 -8879.767,E2 -8879.767} C_VEL
LIN {X 0,Y 448.535,Z 535.778,A -85,B 0,C 180,E1 -8880.683,E2 -8880.683} C_VEL
LIN {X 0,Y 447.928,Z 545.351,A -85,B 0,C 180,E1 -8881.639,E2 -8881.639} C_VEL
LIN {X 0,Y 447.379,Z 553.672,A -85,B 0,C 180,E1 -8882.646,E2 -8882.646} C_VEL
LIN {X 0,Y 446.903,Z 562.02,A -85,B 0,C 180,E1 -8883.876,E2 -8883.876} C_VEL
LIN {X 0,Y 446.371,Z 569.994,A -85,B 0,C 180,E1 -8885.34,E2 -8885.34} C_VEL
LIN {X 0,Y 446.005,Z 576.289,A -85,B 0,C 180,E1 -8886.801,E2 -8886.801} C_VEL
LIN {X 0,Y 445.955,Z 577.114,A -85,B 0,C 180,E1 -8887.029,E2 -8887.029} C_VEL
LIN {X 0,Y 445.159,Z 579.562,A -85,B 0,C 180,E1 -8887.716,E2 -8887.716} C_VEL
LIN {X 0,Y 442.104,Z 583.082,A -85,B 0,C 180,E1 -8888.849,E2 -8888.849} C_VEL
LIN {X 0,Y 439.566,Z 585.361,A -85,B 0,C 180,E1 -8889.784,E2 -8889.784} C_VEL
LIN {X 0,Y 438.461,Z 586.76,A -85,B 0,C 180,E1 -8890.522,E2 -8890.522} C_VEL
LIN {X 0,Y 438.361,Z 587.142,A -85,B 0,C 180,E1 -8890.775,E2 -8890.775} C_VEL
LIN {X 0,Y 438.23,Z 588.843,A -85,B 0,C 180,E1 -8892.26,E2 -8892.26} C_VEL
LIN {X 0,Y 438.197,Z 589.399,A -85,B 0,C 180,E1 -8893.221,E2 -8893.221} C_VEL
LIN {X 0,Y 438.248,Z 589.48,A -85,B 0,C 180,E1 -8894.197,E2 -8894.197} C_VEL
LIN {X 0,Y 438.266,Z 589.16,A -85,B 0,C 180,E1 -8895.133,E2 -8895.133} C_VEL
LIN {X 0,Y 438.263,Z 588.44,A -85,B 0,C 180,E1 -8896.082,E2 -8896.082} C_VEL
LIN {X 0,Y 438.324,Z 587.277,A -85,B 0,C 180,E1 -8897.028,E2 -8897.028} C_VEL
LIN {X 0,Y 438.499,Z 584.725,A -85,B 0,C 180,E1 -8898.443,E2 -8898.443} C_VEL
LIN {X 0,Y 438.621,Z 581.162,A -85,B 0,C 180,E1 -8899.849,E2 -8899.849} C_VEL
LIN {X 0,Y 438.899,Z 576.468,A -85,B 0,C 180,E1 -8901.25,E2 -8901.25} C_VEL
LIN {X 0,Y 439.249,Z 570.013,A -85,B 0,C 180,E1 -8902.753,E2 -8902.753} C_VEL
LIN {X 0,Y 439.622,Z 563.15,A -85,B 0,C 180,E1 -8904.036,E2 -8904.036} C_VEL
LIN {X 0,Y 440.072,Z 555.625,A -85,B 0,C 180,E1 -8905.191,E2 -8905.191} C_VEL
LIN {X 0,Y 440.586,Z 546.533,A -85,B 0,C 180,E1 -8906.342,E2 -8906.342} C_VEL
LIN {X 0,Y 441.203,Z 536.423,A -85,B 0,C 180,E1 -8907.375,E2 -8907.375} C_VEL
LIN {X 0,Y 441.778,Z 525.225,A -85,B 0,C 180,E1 -8908.291,E2 -8908.291} C_VEL
LIN {X 0,Y 442.317,Z 514.598,A -85,B 0,C 180,E1 -8908.976,E2 -8908.976} C_VEL
LIN {X 0,Y 442.679,Z 502.159,A -85,B 0,C 180,E1 -8909.591,E2 -8909.591} C_VEL
LIN {X 0,Y 443.008,Z 489.109,A -85,B 0,C 180,E1 -8910.027,E2 -8910.027} C_VEL
LIN {X 0,Y 443.283,Z 471.074,A -85,B 0,C 180,E1 -8910.367,E2 -8910.367} C_VEL
LIN {X 0,Y 443.928,Z 395.427,A -85,B 0,C 180,E1 -8911.602,E2 -8911.602} C_VEL
LIN {X 0,Y 440.672,Z 379.482,A -85,B 0,C 180,E1 -8911.999,E2 -8911.999} C_VEL
LIN {X 0,Y 440.862,Z 374.337,A -85,B 0,C 180,E1 -8913.198,E2 -8913.198} C_VEL
LIN {X 0,Y 439.531,Z 366.738,A -85,B 0,C 180,E1 -8915.103,E2 -8915.103} C_VEL
LIN {X 0,Y 439.558,Z 366.735,A -85,B 0,C 180,E1 -8917.556,E2 -8917.556} C_VEL
LIN {X 0,Y 439.468,Z 366.739,A -85,B 0,C 180,E1 -8920.132,E2 -8920.132} C_VEL
LIN {X 0,Y 439.471,Z 366.741,A -85,B 0,C 180,E1 -8922.937,E2 -8922.937} C_VEL
LIN {X 0,Y 439.452,Z 366.74,A -85,B 0,C 180,E1 -8926.348,E2 -8926.348} C_VEL
LIN {X 0,Y 439.407,Z 366.75,A -85,B 0,C 180,E1 -8929.626,E2 -8929.626} C_VEL
LIN {X 0,Y 439.369,Z 366.751,A -85,B 0,C 180,E1 -8932.575,E2 -8932.575} C_VEL
LIN {X 0,Y 439.409,Z 366.749,A -85,B 0,C 180,E1 -8935.584,E2 -8935.584} C_VEL
LIN {X 0,Y 439.42,Z 366.746,A -85,B 0,C 180,E1 -8938.673,E2 -8938.673} C_VEL
LIN {X 0,Y 439.386,Z 366.749,A -85,B 0,C 180,E1 -8942.032,E2 -8942.032} C_VEL
LIN {X 0,Y 439.397,Z 366.752,A -85,B 0,C 180,E1 -8945.34,E2 -8945.34} C_VEL
LIN {X 0,Y 439.392,Z 366.75,A -85,B 0,C 180,E1 -8948.593,E2 -8948.593} C_VEL
LIN {X 0,Y 439.387,Z 366.754,A -85,B 0,C 180,E1 -8951.256,E2 -8951.256} C_VEL
LIN {X 0,Y 439.401,Z 366.751,A -85,B 0,C 180,E1 -8954.728,E2 -8954.728} C_VEL
LIN {X 0,Y 439.396,Z 366.748,A -85,B 0,C 180,E1 -8957.795,E2 -8957.795} C_VEL
LIN {X 0,Y 439.434,Z 366.743,A -85,B 0,C 180,E1 -8960.228,E2 -8960.228} C_VEL
LIN {X 0,Y 439.373,Z 366.751,A -85,B 0,C 180,E1 -8963.712,E2 -8963.712} C_VEL
LIN {X 0,Y 439.368,Z 366.757,A -85,B 0,C 180,E1 -8967.053,E2 -8967.053} C_VEL
LIN {X 0,Y 439.377,Z 366.751,A -85,B 0,C 180,E1 -8970.273,E2 -8970.273} C_VEL
LIN {X 0,Y 439.424,Z 366.745,A -85,B 0,C 180,E1 -8973.396,E2 -8973.396} C_VEL
LIN {X 0,Y 439.38,Z 366.753,A -85,B 0,C 180,E1 -8976.429,E2 -8976.429} C_VEL
LIN {X 0,Y 439.381,Z 366.75,A -85,B 0,C 180,E1 -8979.396,E2 -8979.396} C_VEL
LIN {X 0,Y 439.424,Z 366.747,A -85,B 0,C 180,E1 -8982.309,E2 -8982.309} C_VEL
LIN {X 0,Y 439.441,Z 366.744,A -85,B 0,C 180,E1 -8985.173,E2 -8985.173} C_VEL
LIN {X 0,Y 439.476,Z 366.738,A -85,B 0,C 180,E1 -8988.001,E2 -8988.001} C_VEL
LIN {X 0,Y 439.539,Z 366.73,A -85,B 0,C 180,E1 -8991.726,E2 -8991.726} C_VEL
LIN {X 0,Y 439.615,Z 366.727,A -85,B 0,C 180,E1 -8994.495,E2 -8994.495} C_VEL
LIN {X 0,Y 439.627,Z 366.722,A -85,B 0,C 180,E1 -8998.168,E2 -8998.168} C_VEL
LIN {X 0,Y 439.754,Z 366.705,A -85,B 0,C 180,E1 -9000,E2 -9000} C_VEL
LIN {X 0,Y 439.648,Z 366.721,A -85,B 0,C 180,E1 -9002.749,E2 -9002.749} C_VEL
LIN {X 0,Y 439.609,Z 366.729,A -85,B 0,C 180,E1 -9006.425,E2 -9006.425} C_VEL
LIN {X 0,Y 439.492,Z 366.736,A -85,B 0,C 180,E1 -9009.202,E2 -9009.202} C_VEL
LIN {X 0,Y 439.457,Z 366.741,A -85,B 0,C 180,E1 -9012.938,E2 -9012.938} C_VEL
LIN {X 0,Y 439.452,Z 366.748,A -85,B 0,C 180,E1 -9016.355,E2 -9016.355} C_VEL
LIN {X 0,Y 439.394,Z 366.749,A -85,B 0,C 180,E1 -9019.627,E2 -9019.627} C_VEL
LIN {X 0,Y 439.357,Z 366.756,A -85,B 0,C 180,E1 -9022.576,E2 -9022.576} C_VEL
LIN {X 0,Y 439.397,Z 366.748,A -85,B 0,C 180,E1 -9025.585,E2 -9025.585} C_VEL
LIN {X 0,Y 439.418,Z 366.747,A -85,B 0,C 180,E1 -9028.673,E2 -9028.673} C_VEL
LIN {X 0,Y 439.368,Z 366.755,A -85,B 0,C 180,E1 -9031.861,E2 -9031.861} C_VEL
LIN {X 0,Y 439.395,Z 366.748,A -85,B 0,C 180,E1 -9035.156,E2 -9035.156} C_VEL
LIN {X 0,Y 439.393,Z 366.75,A -85,B 0,C 180,E1 -9038.594,E2 -9038.594} C_VEL
LIN {X 0,Y 439.4,Z 366.747,A -85,B 0,C 180,E1 -9041.26,E2 -9041.26} C_VEL
LIN {X 0,Y 439.404,Z 366.747,A -85,B 0,C 180,E1 -9044.729,E2 -9044.729} C_VEL
LIN {X 0,Y 439.394,Z 366.753,A -85,B 0,C 180,E1 -9047.797,E2 -9047.797} C_VEL
LIN {X 0,Y 439.451,Z 366.745,A -85,B 0,C 180,E1 -9050.231,E2 -9050.231} C_VEL
LIN {X 0,Y 439.375,Z 366.755,A -85,B 0,C 180,E1 -9053.714,E2 -9053.714} C_VEL
LIN {X 0,Y 439.374,Z 366.75,A -85,B 0,C 180,E1 -9057.055,E2 -9057.055} C_VEL
LIN {X 0,Y 439.396,Z 366.756,A -85,B 0,C 180,E1 -9060.276,E2 -9060.276} C_VEL
LIN {X 0,Y 439.516,Z 366.862,A -85,B 0,C 180,E1 -9062.632,E2 -9062.632} C_VEL
LIN {X 0,Y 442.142,Z 380.509,A -85,B 0,C 180,E1 -9065.319,E2 -9065.319} C_VEL
LIN {X 0,Y 441.7,Z 391.65,A -85,B 0,C 180,E1 -9067.347,E2 -9067.347} C_VEL
LIN {X 0,Y 440.699,Z 410.209,A -85,B 0,C 180,E1 -9070.677,E2 -9070.677} C_VEL
LIN {X 0,Y 440.331,Z 417.617,A -85,B 0,C 180,E1 -9071.994,E2 -9071.994} C_VEL
LIN {X 0,Y 443.723,Z 441.024,A -85,B 0,C 180,E1 -9072.513,E2 -9072.513} C_VEL
LIN {X 0,Y 442.945,Z 526.992,A -85,B 0,C 180,E1 -9073.939,E2 -9073.939} C_VEL
LIN {X 0,Y 442.441,Z 540.791,A -85,B 0,C 180,E1 -9074.363,E2 -9074.363} C_VEL
LIN {X 0,Y 441.905,Z 553.704,A -85,B 0,C 180,E1 -9074.964,E2 -9074.964} C_VEL
LIN {X 0,Y 441.246,Z 565.486,A -85,B 0,C 180,E1 -9075.708,E2 -9075.708} C_VEL
LIN {X 0,Y 440.591,Z 577.256,A -85,B 0,C 180,E1 -9076.663,E2 -9076.663} C_VEL
LIN {X 0,Y 440.085,Z 588.094,A -85,B 0,C 180,E1 -9077.784,E2 -9077.784} C_VEL
LIN {X 0,Y 439.54,Z 597.146,A -85,B 0,C 180,E1 -9078.938,E2 -9078.938} C_VEL
LIN {X 0,Y 439.015,Z 605.983,A -85,B 0,C 180,E1 -9080.323,E2 -9080.323} C_VEL
LIN {X 0,Y 438.696,Z 613.038,A -85,B 0,C 180,E1 -9081.71,E2 -9081.71} C_VEL
LIN {X 0,Y 438.494,Z 618.682,A -85,B 0,C 180,E1 -9083.096,E2 -9083.096} C_VEL
LIN {X 0,Y 438.386,Z 623.115,A -85,B 0,C 180,E1 -9084.48,E2 -9084.48} C_VEL
LIN {X 0,Y 438.348,Z 625.455,A -85,B 0,C 180,E1 -9085.402,E2 -9085.402} C_VEL
LIN {X 0,Y 438.298,Z 627.361,A -85,B 0,C 180,E1 -9086.323,E2 -9086.323} C_VEL
LIN {X 0,Y 438.372,Z 628.814,A -85,B 0,C 180,E1 -9087.243,E2 -9087.243} C_VEL
LIN {X 0,Y 438.305,Z 630.464,A -85,B 0,C 180,E1 -9089.081,E2 -9089.081} C_VEL
LIN {X 0,Y 438.309,Z 630.706,A -85,B 0,C 180,E1 -9090,E2 -9090} C_VEL
LIN {X 0,Y 438.305,Z 630.523,A -85,B 0,C 180,E1 -9090.919,E2 -9090.919} C_VEL
LIN {X 0,Y 438.372,Z 628.946,A -85,B 0,C 180,E1 -9092.757,E2 -9092.757} C_VEL
LIN {X 0,Y 438.293,Z 627.56,A -85,B 0,C 180,E1 -9093.677,E2 -9093.677} C_VEL
LIN {X 0,Y 438.39,Z 624.647,A -85,B 0,C 180,E1 -9095.058,E2 -9095.058} C_VEL
LIN {X 0,Y 438.447,Z 620.7,A -85,B 0,C 180,E1 -9096.442,E2 -9096.442} C_VEL
LIN {X 0,Y 438.639,Z 615.625,A -85,B 0,C 180,E1 -9097.827,E2 -9097.827} C_VEL
LIN {X 0,Y 438.914,Z 609.259,A -85,B 0,C 180,E1 -9099.214,E2 -9099.214} C_VEL
LIN {X 0,Y 439.344,Z 601.304,A -85,B 0,C 180,E1 -9100.6,E2 -9100.6} C_VEL
LIN {X 0,Y 439.891,Z 593.231,A -85,B 0,C 180,E1 -9101.753,E2 -9101.753} C_VEL
LIN {X 0,Y 440.485,Z 583.402,A -85,B 0,C 180,E1 -9102.907,E2 -9102.907} C_VEL
LIN {X 0,Y 441.136,Z 572.454,A -85,B 0,C 180,E1 -9103.943,E2 -9103.943} C_VEL
LIN {X 0,Y 441.9,Z 559.983,A -85,B 0,C 180,E1 -9104.859,E2 -9104.859} C_VEL
LIN {X 0,Y 442.591,Z 547.754,A -85,B 0,C 180,E1 -9105.543,E2 -9105.543} C_VEL
LIN {X 0,Y 443.11,Z 534.907,A -85,B 0,C 180,E1 -9106.055,E2 -9106.055} C_VEL
LIN {X 0,Y 443.489,Z 521.33,A -85,B 0,C 180,E1 -9106.396,E2 -9106.396} C_VEL
LIN {X 0,Y 444.225,Z 440.613,A -85,B 0,C 180,E1 -9107.73,E2 -9107.73} C_VEL
LIN {X 0,Y 440.564,Z 417.21,A -85,B 0,C 180,E1 -9108.307,E2 -9108.307} C_VEL
LIN {X 0,Y 441.629,Z 398.503,A -85,B 0,C 180,E1 -9111.715,E2 -9111.715} C_VEL
LIN {X 0,Y 442.534,Z 384.082,A -85,B 0,C 180,E1 -9114.387,E2 -9114.387} C_VEL
LIN {X 0,Y 442.314,Z 380.502,A -85,B 0,C 180,E1 -9115.085,E2 -9115.085} C_VEL
LIN {X 0,Y 440.154,Z 369.617,A -85,B 0,C 180,E1 -9117.342,E2 -9117.342} C_VEL
LIN {X 0,Y 439.449,Z 366.746,A -85,B 0,C 180,E1 -9117.987,E2 -9117.987} C_VEL
LIN {X 0,Y 439.365,Z 366.755,A -85,B 0,C 180,E1 -9120.787,E2 -9120.787} C_VEL
LIN {X 0,Y 439.386,Z 366.754,A -85,B 0,C 180,E1 -9124.043,E2 -9124.043} C_VEL
LIN {X 0,Y 439.362,Z 366.756,A -85,B 0,C 180,E1 -9127.433,E2 -9127.433} C_VEL
LIN {X 0,Y 439.428,Z 366.749,A -85,B 0,C 180,E1 -9129.853,E2 -9129.853} C_VEL
LIN {X 0,Y 439.378,Z 366.75,A -85,B 0,C 180,E1 -9132.626,E2 -9132.626} C_VEL
LIN {X 0,Y 439.398,Z 366.755,A -85,B 0,C 180,E1 -9136.033,E2 -9136.033} C_VEL
LIN {X 0,Y 439.395,Z 366.75,A -85,B 0,C 180,E1 -9139.021,E2 -9139.021} C_VEL
LIN {X 0,Y 439.387,Z 366.754,A -85,B 0,C 180,E1 -9141.604,E2 -9141.604} C_VEL
LIN {X 0,Y 439.395,Z 366.749,A -85,B 0,C 180,E1 -9144.844,E2 -9144.844} C_VEL
LIN {X 0,Y 439.368,Z 366.754,A -85,B 0,C 180,E1 -9148.139,E2 -9148.139} C_VEL
LIN {X 0,Y 439.418,Z 366.746,A -85,B 0,C 180,E1 -9151.327,E2 -9151.327} C_VEL
LIN {X 0,Y 439.397,Z 366.746,A -85,B 0,C 180,E1 -9154.415,E2 -9154.415} C_VEL
LIN {X 0,Y 439.357,Z 366.757,A -85,B 0,C 180,E1 -9157.424,E2 -9157.424} C_VEL
LIN {X 0,Y 439.433,Z 366.744,A -85,B 0,C 180,E1 -9160.662,E2 -9160.662} C_VEL
LIN {X 0,Y 439.467,Z 366.74,A -85,B 0,C 180,E1 -9164.225,E2 -9164.225} C_VEL
LIN {X 0,Y 439.475,Z 366.738,A -85,B 0,C 180,E1 -9168.001,E2 -9168.001} C_VEL
LIN {X 0,Y 439.539,Z 366.728,A -85,B 0,C 180,E1 -9171.726,E2 -9171.726} C_VEL
LIN {X 0,Y 439.613,Z 366.721,A -85,B 0,C 180,E1 -9174.496,E2 -9174.496} C_VEL
LIN {X 0,Y 439.627,Z 366.716,A -85,B 0,C 180,E1 -9178.168,E2 -9178.168} C_VEL
LIN {X 0,Y 439.756,Z 366.705,A -85,B 0,C 180,E1 -9180,E2 -9180} C_VEL
LIN {X 0,Y 439.649,Z 366.713,A -85,B 0,C 180,E1 -9182.749,E2 -9182.749} C_VEL
LIN {X 0,Y 439.611,Z 366.72,A -85,B 0,C 180,E1 -9186.426,E2 -9186.426} C_VEL
LIN {X 0,Y 439.493,Z 366.742,A -85,B 0,C 180,E1 -9189.202,E2 -9189.202} C_VEL
LIN {X 0,Y 439.461,Z 366.74,A -85,B 0,C 180,E1 -9192.938,E2 -9192.938} C_VEL
LIN {X 0,Y 439.44,Z 366.739,A -85,B 0,C 180,E1 -9196.349,E2 -9196.349} C_VEL
LIN {X 0,Y 439.427,Z 366.743,A -85,B 0,C 180,E1 -9199.625,E2 -9199.625} C_VEL
LIN {X 0,Y 439.367,Z 366.755,A -85,B 0,C 180,E1 -9202.576,E2 -9202.576} C_VEL
LIN {X 0,Y 439.4,Z 366.75,A -85,B 0,C 180,E1 -9205.586,E2 -9205.586} C_VEL
LIN {X 0,Y 439.412,Z 366.75,A -85,B 0,C 180,E1 -9208.674,E2 -9208.674} C_VEL
LIN {X 0,Y 439.365,Z 366.754,A -85,B 0,C 180,E1 -9212.031,E2 -9212.031} C_VEL
LIN {X 0,Y 439.392,Z 366.751,A -85,B 0,C 180,E1 -9215.342,E2 -9215.342} C_VEL
LIN {X 0,Y 439.393,Z 366.753,A -85,B 0,C 180,E1 -9218.594,E2 -9218.594} C_VEL
LIN {X 0,Y 439.402,Z 366.748,A -85,B 0,C 180,E1 -9221.26,E2 -9221.26} C_VEL
LIN {X 0,Y 439.408,Z 366.75,A -85,B 0,C 180,E1 -9224.729,E2 -9224.729} C_VEL
LIN {X 0,Y 439.397,Z 366.749,A -85,B 0,C 180,E1 -9227.797,E2 -9227.797} C_VEL
LIN {X 0,Y 439.436,Z 366.75,A -85,B 0,C 180,E1 -9230.23,E2 -9230.23} C_VEL
LIN {X 0,Y 439.397,Z 366.816,A -85,B 0,C 180,E1 -9232.462,E2 -9232.462} C_VEL
LIN {X 0,Y 441.037,Z 375.455,A -85,B 0,C 180,E1 -9234.7,E2 -9234.7} C_VEL
LIN {X 0,Y 441.046,Z 380.14,A -85,B 0,C 180,E1 -9235.788,E2 -9235.788} C_VEL
LIN {X 0,Y 444.693,Z 396.276,A -85,B 0,C 180,E1 -9236.24,E2 -9236.24} C_VEL
LIN {X 0,Y 443.67,Z 486.648,A -85,B 0,C 180,E1 -9237.75,E2 -9237.75} C_VEL
LIN {X 0,Y 443.268,Z 500.184,A -85,B 0,C 180,E1 -9238.169,E2 -9238.169} C_VEL
LIN {X 0,Y 442.911,Z 511.922,A -85,B 0,C 180,E1 -9238.711,E2 -9238.711} C_VEL
LIN {X 0,Y 442.351,Z 523.772,A -85,B 0,C 180,E1 -9239.443,E2 -9239.443} C_VEL
LIN {X 0,Y 441.776,Z 534.759,A -85,B 0,C 180,E1 -9240.321,E2 -9240.321} C_VEL
LIN {X 0,Y 441.1,Z 544.65,A -85,B 0,C 180,E1 -9241.299,E2 -9241.299} C_VEL
LIN {X 0,Y 440.454,Z 554.018,A -85,B 0,C 180,E1 -9242.437,E2 -9242.437} C_VEL
LIN {X 0,Y 439.951,Z 562.356,A -85,B 0,C 180,E1 -9243.687,E2 -9243.687} C_VEL
LIN {X 0,Y 439.388,Z 570.323,A -85,B 0,C 180,E1 -9245.174,E2 -9245.174} C_VEL
LIN {X 0,Y 439.05,Z 575.659,A -85,B 0,C 180,E1 -9246.411,E2 -9246.411} C_VEL
LIN {X 0,Y 438.731,Z 580.734,A -85,B 0,C 180,E1 -9247.887,E2 -9247.887} C_VEL
LIN {X 0,Y 438.526,Z 584.544,A -85,B 0,C 180,E1 -9249.355,E2 -9249.355} C_VEL
LIN {X 0,Y 438.361,Z 587.142,A -85,B 0,C 180,E1 -9250.775,E2 -9250.775} C_VEL
LIN {X 0,Y 437.647,Z 588.194,A -85,B 0,C 180,E1 -9251.528,E2 -9251.528} C_VEL
LIN {X 0,Y 434.711,Z 589.349,A -85,B 0,C 180,E1 -9252.762,E2 -9252.762} C_VEL
LIN {X 0,Y 432.26,Z 589.777,A -85,B 0,C 180,E1 -9253.764,E2 -9253.764} C_VEL
LIN {X 0,Y 431.229,Z 589.744,A -85,B 0,C 180,E1 -9254.539,E2 -9254.539} C_VEL
LIN {X 0,Y 431.156,Z 589.641,A -85,B 0,C 180,E1 -9254.802,E2 -9254.802} C_VEL
LIN {X 0,Y 431.162,Z 588.98,A -85,B 0,C 180,E1 -9255.848,E2 -9255.848} C_VEL
LIN {X 0,Y 431.227,Z 587.938,A -85,B 0,C 180,E1 -9256.811,E2 -9256.811} C_VEL
LIN {X 0,Y 431.352,Z 586.31,A -85,B 0,C 180,E1 -9257.847,E2 -9257.847} C_VEL
LIN {X 0,Y 431.489,Z 583.402,A -85,B 0,C 180,E1 -9259.204,E2 -9259.204} C_VEL
LIN {X 0,Y 431.676,Z 579.287,A -85,B 0,C 180,E1 -9260.63,E2 -9260.63} C_VEL
LIN {X 0,Y 432.054,Z 572.972,A -85,B 0,C 180,E1 -9262.288,E2 -9262.288} C_VEL
LIN {X 0,Y 432.407,Z 566.125,A -85,B 0,C 180,E1 -9263.702,E2 -9263.702} C_VEL
LIN {X 0,Y 432.888,Z 559.117,A -85,B 0,C 180,E1 -9264.877,E2 -9264.877} C_VEL
LIN {X 0,Y 433.396,Z 550.7,A -85,B 0,C 180,E1 -9266.048,E2 -9266.048} C_VEL
LIN {X 0,Y 434.035,Z 540.293,A -85,B 0,C 180,E1 -9267.216,E2 -9267.216} C_VEL
LIN {X 0,Y 434.645,Z 529.992,A -85,B 0,C 180,E1 -9268.147,E2 -9268.147} C_VEL
LIN {X 0,Y 435.269,Z 518.702,A -85,B 0,C 180,E1 -9268.959,E2 -9268.959} C_VEL
LIN {X 0,Y 435.699,Z 507.105,A -85,B 0,C 180,E1 -9269.602,E2 -9269.602} C_VEL
LIN {X 0,Y 436.085,Z 494.963,A -85,B 0,C 180,E1 -9270.086,E2 -9270.086} C_VEL
LIN {X 0,Y 436.335,Z 482.251,A -85,B 0,C 180,E1 -9270.414,E2 -9270.414} C_VEL
LIN {X 0,Y 437.238,Z 397.087,A -85,B 0,C 180,E1 -9271.824,E2 -9271.824} C_VEL
LIN {X 0,Y 433.727,Z 379.822,A -85,B 0,C 180,E1 -9272.258,E2 -9272.258} C_VEL
LIN {X 0,Y 433.9,Z 375.601,A -85,B 0,C 180,E1 -9273.25,E2 -9273.25} C_VEL
LIN {X 0,Y 432.54,Z 367.609,A -85,B 0,C 180,E1 -9275.302,E2 -9275.302} C_VEL
LIN {X 0,Y 432.469,Z 367.614,A -85,B 0,C 180,E1 -9278.41,E2 -9278.41} C_VEL
LIN {X 0,Y 432.464,Z 367.611,A -85,B 0,C 180,E1 -9282.196,E2 -9282.196} C_VEL
LIN {X 0,Y 432.435,Z 367.615,A -85,B 0,C 180,E1 -9286.038,E2 -9286.038} C_VEL
LIN {X 0,Y 432.391,Z 367.626,A -85,B 0,C 180,E1 -9289.485,E2 -9289.485} C_VEL
LIN {X 0,Y 432.323,Z 367.632,A -85,B 0,C 180,E1 -9292.963,E2 -9292.963} C_VEL
LIN {X 0,Y 432.367,Z 367.623,A -85,B 0,C 180,E1 -9296.032,E2 -9296.032} C_VEL
LIN {X 0,Y 432.346,Z 367.634,A -85,B 0,C 180,E1 -9299.186,E2 -9299.186} C_VEL
LIN {X 0,Y 432.334,Z 367.627,A -85,B 0,C 180,E1 -9302.294,E2 -9302.294} C_VEL
LIN {X 0,Y 432.342,Z 367.629,A -85,B 0,C 180,E1 -9304.676,E2 -9304.676} C_VEL
LIN {X 0,Y 432.349,Z 367.625,A -85,B 0,C 180,E1 -9308.148,E2 -9308.148} C_VEL
LIN {X 0,Y 432.331,Z 367.629,A -85,B 0,C 180,E1 -9311.601,E2 -9311.601} C_VEL
LIN {X 0,Y 432.332,Z 367.628,A -85,B 0,C 180,E1 -9314.346,E2 -9314.346} C_VEL
LIN {X 0,Y 432.323,Z 367.636,A -85,B 0,C 180,E1 -9317.014,E2 -9317.014} C_VEL
LIN {X 0,Y 432.339,Z 367.627,A -85,B 0,C 180,E1 -9319.818,E2 -9319.818} C_VEL
LIN {X 0,Y 432.312,Z 367.637,A -85,B 0,C 180,E1 -9323.022,E2 -9323.022} C_VEL
LIN {X 0,Y 432.355,Z 367.625,A -85,B 0,C 180,E1 -9325.996,E2 -9325.996} C_VEL
LIN {X 0,Y 432.342,Z 367.627,A -85,B 0,C 180,E1 -9329.489,E2 -9329.489} C_VEL
LIN {X 0,Y 432.387,Z 367.627,A -85,B 0,C 180,E1 -9332.927,E2 -9332.927} C_VEL
LIN {X 0,Y 432.365,Z 367.624,A -85,B 0,C 180,E1 -9336.023,E2 -9336.023} C_VEL
LIN {X 0,Y 432.343,Z 367.63,A -85,B 0,C 180,E1 -9339.045,E2 -9339.045} C_VEL
LIN {X 0,Y 432.37,Z 367.623,A -85,B 0,C 180,E1 -9342.01,E2 -9342.01} C_VEL
LIN {X 0,Y 432.389,Z 367.625,A -85,B 0,C 180,E1 -9344.926,E2 -9344.926} C_VEL
LIN {X 0,Y 432.451,Z 367.613,A -85,B 0,C 180,E1 -9347.803,E2 -9347.803} C_VEL
LIN {X 0,Y 432.484,Z 367.609,A -85,B 0,C 180,E1 -9351.59,E2 -9351.59} C_VEL
LIN {X 0,Y 432.592,Z 367.6,A -85,B 0,C 180,E1 -9354.406,E2 -9354.406} C_VEL
LIN {X 0,Y 432.597,Z 367.597,A -85,B 0,C 180,E1 -9358.138,E2 -9358.138} C_VEL
LIN {X 0,Y 432.724,Z 367.58,A -85,B 0,C 180,E1 -9360,E2 -9360} C_VEL
LIN {X 0,Y 432.597,Z 367.598,A -85,B 0,C 180,E1 -9362.793,E2 -9362.793} C_VEL
LIN {X 0,Y 432.563,Z 367.605,A -85,B 0,C 180,E1 -9366.53,E2 -9366.53} C_VEL
LIN {X 0,Y 432.435,Z 367.615,A -85,B 0,C 180,E1 -9369.353,E2 -9369.353} C_VEL
LIN {X 0,Y 432.422,Z 367.619,A -85,B 0,C 180,E1 -9372.804,E2 -9372.804} C_VEL
LIN {X 0,Y 432.414,Z 367.623,A -85,B 0,C 180,E1 -9376.484,E2 -9376.484} C_VEL
LIN {X 0,Y 432.331,Z 367.631,A -85,B 0,C 180,E1 -9379.961,E2 -9379.961} C_VEL
LIN {X 0,Y 432.311,Z 367.631,A -85,B 0,C 180,E1 -9382.965,E2 -9382.965} C_VEL
LIN {X 0,Y 432.357,Z 367.629,A -85,B 0,C 180,E1 -9386.033,E2 -9386.033} C_VEL
LIN {X 0,Y 432.345,Z 367.626,A -85,B 0,C 180,E1 -9389.187,E2 -9389.187} C_VEL
LIN {X 0,Y 432.319,Z 367.635,A -85,B 0,C 180,E1 -9392.294,E2 -9392.294} C_VEL
LIN {X 0,Y 432.335,Z 367.629,A -85,B 0,C 180,E1 -9394.678,E2 -9394.678} C_VEL
LIN {X 0,Y 432.348,Z 367.633,A -85,B 0,C 180,E1 -9398.149,E2 -9398.149} C_VEL
LIN {X 0,Y 432.368,Z 367.625,A -85,B 0,C 180,E1 -9401.609,E2 -9401.609} C_VEL
LIN {X 0,Y 432.374,Z 367.626,A -85,B 0,C 180,E1 -9404.342,E2 -9404.342} C_VEL
LIN {X 0,Y 432.363,Z 367.626,A -85,B 0,C 180,E1 -9408.394,E2 -9408.394} C_VEL
LIN {X 0,Y 432.352,Z 367.632,A -85,B 0,C 180,E1 -9411.853,E2 -9411.853} C_VEL
LIN {X 0,Y 432.339,Z 367.628,A -85,B 0,C 180,E1 -9415.324,E2 -9415.324} C_VEL
LIN {X 0,Y 432.329,Z 367.628,A -85,B 0,C 180,E1 -9418.655,E2 -9418.655} C_VEL
LIN {X 0,Y 432.449,Z 367.622,A -85,B 0,C 180,E1 -9422.146,E2 -9422.146} C_VEL
LIN {X 0,Y 432.46,Z 367.647,A -85,B 0,C 180,E1 -9422.41,E2 -9422.41} C_VEL
LIN {X 0,Y 435.121,Z 381.452,A -85,B 0,C 180,E1 -9425.169,E2 -9425.169} C_VEL
LIN {X 0,Y 435.023,Z 388.344,A -85,B 0,C 180,E1 -9426.457,E2 -9426.457} C_VEL
LIN {X 0,Y 433.807,Z 408.37,A -85,B 0,C 180,E1 -9430.11,E2 -9430.11} C_VEL
LIN {X 0,Y 433.383,Z 417.278,A -85,B 0,C 180,E1 -9431.725,E2 -9431.725} C_VEL
LIN {X 0,Y 436.898,Z 442.533,A -85,B 0,C 180,E1 -9432.293,E2 -9432.293} C_VEL
LIN {X 0,Y 436.081,Z 526.582,A -85,B 0,C 180,E1 -9433.709,E2 -9433.709} C_VEL
LIN {X 0,Y 435.558,Z 540.406,A -85,B 0,C 180,E1 -9434.14,E2 -9434.14} C_VEL
LIN {X 0,Y 435.037,Z 552.833,A -85,B 0,C 180,E1 -9434.721,E2 -9434.721} C_VEL
LIN {X 0,Y 434.336,Z 564.733,A -85,B 0,C 180,E1 -9435.475,E2 -9435.475} C_VEL
LIN {X 0,Y 433.702,Z 575.961,A -85,B 0,C 180,E1 -9436.389,E2 -9436.389} C_VEL
LIN {X 0,Y 433.107,Z 586.526,A -85,B 0,C 180,E1 -9437.465,E2 -9437.465} C_VEL
LIN {X 0,Y 432.513,Z 596.622,A -85,B 0,C 180,E1 -9438.756,E2 -9438.756} C_VEL
LIN {X 0,Y 431.974,Z 605.503,A -85,B 0,C 180,E1 -9440.164,E2 -9440.164} C_VEL
LIN {X 0,Y 431.64,Z 612.6,A -85,B 0,C 180,E1 -9441.574,E2 -9441.574} C_VEL
LIN {X 0,Y 431.414,Z 618.269,A -85,B 0,C 180,E1 -9442.982,E2 -9442.982} C_VEL
LIN {X 0,Y 431.289,Z 622.72,A -85,B 0,C 180,E1 -9444.389,E2 -9444.389} C_VEL
LIN {X 0,Y 431.28,Z 625.071,A -85,B 0,C 180,E1 -9445.327,E2 -9445.327} C_VEL
LIN {X 0,Y 431.203,Z 626.984,A -85,B 0,C 180,E1 -9446.262,E2 -9446.262} C_VEL
LIN {X 0,Y 431.281,Z 628.453,A -85,B 0,C 180,E1 -9447.198,E2 -9447.198} C_VEL
LIN {X 0,Y 431.24,Z 629.482,A -85,B 0,C 180,E1 -9448.132,E2 -9448.132} C_VEL
LIN {X 0,Y 431.22,Z 630.368,A -85,B 0,C 180,E1 -9450,E2 -9450} C_VEL
LIN {X 0,Y 431.219,Z 630.2,A -85,B 0,C 180,E1 -9450.934,E2 -9450.934} C_VEL
LIN {X 0,Y 431.28,Z 628.636,A -85,B 0,C 180,E1 -9452.802,E2 -9452.802} C_VEL
LIN {X 0,Y 431.199,Z 627.258,A -85,B 0,C 180,E1 -9453.738,E2 -9453.738} C_VEL
LIN {X 0,Y 431.301,Z 624.362,A -85,B 0,C 180,E1 -9455.142,E2 -9455.142} C_VEL
LIN {X 0,Y 431.375,Z 620.436,A -85,B 0,C 180,E1 -9456.548,E2 -9456.548} C_VEL
LIN {X 0,Y 431.56,Z 615.385,A -85,B 0,C 180,E1 -9457.956,E2 -9457.956} C_VEL
LIN {X 0,Y 431.857,Z 609.056,A -85,B 0,C 180,E1 -9459.366,E2 -9459.366} C_VEL
LIN {X 0,Y 432.35,Z 601.151,A -85,B 0,C 180,E1 -9460.774,E2 -9460.774} C_VEL
LIN {X 0,Y 433.077,Z 591.326,A -85,B 0,C 180,E1 -9462.179,E2 -9462.179} C_VEL
LIN {X 0,Y 433.684,Z 581.146,A -85,B 0,C 180,E1 -9463.349,E2 -9463.349} C_VEL
LIN {X 0,Y 434.448,Z 569.619,A -85,B 0,C 180,E1 -9464.401,E2 -9464.401} C_VEL
LIN {X 0,Y 435.137,Z 558.319,A -85,B 0,C 180,E1 -9465.216,E2 -9465.216} C_VEL
LIN {X 0,Y 435.83,Z 546.82,A -85,B 0,C 180,E1 -9465.85,E2 -9465.85} C_VEL
LIN {X 0,Y 436.405,Z 533.659,A -85,B 0,C 180,E1 -9466.369,E2 -9466.369} C_VEL
LIN {X 0,Y 436.741,Z 521.003,A -85,B 0,C 180,E1 -9466.686,E2 -9466.686} C_VEL
LIN {X 0,Y 437.558,Z 441.601,A -85,B 0,C 180,E1 -9468.019,E2 -9468.019} C_VEL
LIN {X 0,Y 433.918,Z 418.568,A -85,B 0,C 180,E1 -9468.595,E2 -9468.595} C_VEL
LIN {X 0,Y 433.645,Z 416.76,A -85,B 0,C 180,E1 -9468.664,E2 -9468.664} C_VEL
LIN {X 0,Y 434.772,Z 398.39,A -85,B 0,C 180,E1 -9472.075,E2 -9472.075} C_VEL
LIN {X 0,Y 435.677,Z 384.011,A -85,B 0,C 180,E1 -9474.797,E2 -9474.797} C_VEL
LIN {X 0,Y 433.786,Z 373.512,A -85,B 0,C 180,E1 -9476.99,E2 -9476.99} C_VEL
LIN {X 0,Y 432.41,Z 367.624,A -85,B 0,C 180,E1 -9478.294,E2 -9478.294} C_VEL
LIN {X 0,Y 432.329,Z 367.63,A -85,B 0,C 180,E1 -9481.345,E2 -9481.345} C_VEL
LIN {X 0,Y 432.339,Z 367.63,A -85,B 0,C 180,E1 -9484.676,E2 -9484.676} C_VEL
LIN {X 0,Y 432.352,Z 367.626,A -85,B 0,C 180,E1 -9488.147,E2 -9488.147} C_VEL
LIN {X 0,Y 432.363,Z 367.625,A -85,B 0,C 180,E1 -9491.606,E2 -9491.606} C_VEL
LIN {X 0,Y 432.374,Z 367.626,A -85,B 0,C 180,E1 -9495.658,E2 -9495.658} C_VEL
LIN {X 0,Y 432.368,Z 367.627,A -85,B 0,C 180,E1 -9498.391,E2 -9498.391} C_VEL
LIN {X 0,Y 432.348,Z 367.633,A -85,B 0,C 180,E1 -9501.851,E2 -9501.851} C_VEL
LIN {X 0,Y 432.335,Z 367.631,A -85,B 0,C 180,E1 -9505.322,E2 -9505.322} C_VEL
LIN {X 0,Y 432.317,Z 367.63,A -85,B 0,C 180,E1 -9508.654,E2 -9508.654} C_VEL
LIN {X 0,Y 432.374,Z 367.624,A -85,B 0,C 180,E1 -9511.368,E2 -9511.368} C_VEL
LIN {X 0,Y 432.357,Z 367.625,A -85,B 0,C 180,E1 -9513.967,E2 -9513.967} C_VEL
LIN {X 0,Y 432.311,Z 367.632,A -85,B 0,C 180,E1 -9517.035,E2 -9517.035} C_VEL
LIN {X 0,Y 432.378,Z 367.623,A -85,B 0,C 180,E1 -9520.514,E2 -9520.514} C_VEL
LIN {X 0,Y 432.434,Z 367.618,A -85,B 0,C 180,E1 -9523.961,E2 -9523.961} C_VEL
LIN {X 0,Y 432.451,Z 367.613,A -85,B 0,C 180,E1 -9527.803,E2 -9527.803} C_VEL
LIN {X 0,Y 432.483,Z 367.608,A -85,B 0,C 180,E1 -9531.59,E2 -9531.59} C_VEL
LIN {X 0,Y 432.589,Z 367.596,A -85,B 0,C 180,E1 -9534.406,E2 -9534.406} C_VEL
LIN {X 0,Y 432.597,Z 367.592,A -85,B 0,C 180,E1 -9538.138,E2 -9538.138} C_VEL
LIN {X 0,Y 432.726,Z 367.58,A -85,B 0,C 180,E1 -9540,E2 -9540} C_VEL
LIN {X 0,Y 432.599,Z 367.591,A -85,B 0,C 180,E1 -9542.794,E2 -9542.794} C_VEL
LIN {X 0,Y 432.566,Z 367.598,A -85,B 0,C 180,E1 -9546.531,E2 -9546.531} C_VEL
LIN {X 0,Y 432.436,Z 367.621,A -85,B 0,C 180,E1 -9549.354,E2 -9549.354} C_VEL
LIN {X 0,Y 432.424,Z 367.615,A -85,B 0,C 180,E1 -9552.805,E2 -9552.805} C_VEL
LIN {X 0,Y 432.405,Z 367.616,A -85,B 0,C 180,E1 -9556.48,E2 -9556.48} C_VEL
LIN {X 0,Y 432.373,Z 367.62,A -85,B 0,C 180,E1 -9559.959,E2 -9559.959} C_VEL
LIN {X 0,Y 432.318,Z 367.635,A -85,B 0,C 180,E1 -9562.965,E2 -9562.965} C_VEL
LIN {X 0,Y 432.359,Z 367.626,A -85,B 0,C 180,E1 -9566.033,E2 -9566.033} C_VEL
LIN {X 0,Y 432.337,Z 367.632,A -85,B 0,C 180,E1 -9569.188,E2 -9569.188} C_VEL
LIN {X 0,Y 432.318,Z 367.634,A -85,B 0,C 180,E1 -9572.444,E2 -9572.444} C_VEL
LIN {X 0,Y 432.341,Z 367.628,A -85,B 0,C 180,E1 -9575.633,E2 -9575.633} C_VEL
LIN {X 0,Y 432.355,Z 367.632,A -85,B 0,C 180,E1 -9578.718,E2 -9578.718} C_VEL
LIN {X 0,Y 432.371,Z 367.622,A -85,B 0,C 180,E1 -9581.793,E2 -9581.793} C_VEL
LIN {X 0,Y 432.376,Z 367.628,A -85,B 0,C 180,E1 -9584.342,E2 -9584.342} C_VEL
LIN {X 0,Y 432.334,Z 367.631,A -85,B 0,C 180,E1 -9588.204,E2 -9588.204} C_VEL
LIN {X 0,Y 432.353,Z 367.633,A -85,B 0,C 180,E1 -9591.284,E2 -9591.284} C_VEL
LIN {X 0,Y 432.376,Z 367.778,A -85,B 0,C 180,E1 -9592.217,E2 -9592.217} C_VEL
LIN {X 0,Y 434.148,Z 376.994,A -85,B 0,C 180,E1 -9594.641,E2 -9594.641} C_VEL
LIN {X 0,Y 434.187,Z 380.41,A -85,B 0,C 180,E1 -9595.448,E2 -9595.448} C_VEL
LIN {X 0,Y 438.037,Z 397.396,A -85,B 0,C 180,E1 -9595.938,E2 -9595.938} C_VEL
LIN {X 0,Y 436.935,Z 487.187,A -85,B 0,C 180,E1 -9597.464,E2 -9597.464} C_VEL
LIN {X 0,Y 436.517,Z 501.065,A -85,B 0,C 180,E1 -9597.907,E2 -9597.907} C_VEL
LIN {X 0,Y 436.089,Z 513.262,A -85,B 0,C 180,E1 -9598.49,E2 -9598.49} C_VEL
LIN {X 0,Y 435.433,Z 525.844,A -85,B 0,C 180,E1 -9599.308,E2 -9599.308} C_VEL
LIN {X 0,Y 434.849,Z 536.517,A -85,B 0,C 180,E1 -9600.201,E2 -9600.201} C_VEL
LIN {X 0,Y 434.131,Z 546.313,A -85,B 0,C 180,E1 -9601.21,E2 -9601.21} C_VEL
LIN {X 0,Y 433.44,Z 556.168,A -85,B 0,C 180,E1 -9602.477,E2 -9602.477} C_VEL
LIN {X 0,Y 432.856,Z 564.305,A -85,B 0,C 180,E1 -9603.769,E2 -9603.769} C_VEL
LIN {X 0,Y 432.293,Z 572.265,A -85,B 0,C 180,E1 -9605.346,E2 -9605.346} C_VEL
LIN {X 0,Y 431.966,Z 576.961,A -85,B 0,C 180,E1 -9606.509,E2 -9606.509} C_VEL
LIN {X 0,Y 431.64,Z 582.17,A -85,B 0,C 180,E1 -9608.139,E2 -9608.139} C_VEL
LIN {X 0,Y 431.447,Z 585.426,A -85,B 0,C 180,E1 -9609.5,E2 -9609.5} C_VEL
LIN {X 0,Y 431.265,Z 587.913,A -85,B 0,C 180,E1 -9610.979,E2 -9610.979} C_VEL
LIN {X 0,Y 431.192,Z 588.974,A -85,B 0,C 180,E1 -9611.96,E2 -9611.96} C_VEL
LIN {X 0,Y 431.125,Z 589.619,A -85,B 0,C 180,E1 -9612.937,E2 -9612.937} C_VEL
LIN {X 0,Y 431.161,Z 589.828,A -85,B 0,C 180,E1 -9614.096,E2 -9614.096} C_VEL
LIN {X 0,Y 431.156,Z 589.641,A -85,B 0,C 180,E1 -9614.802,E2 -9614.802} C_VEL
LIN {X 0,Y 430.52,Z 589.296,A -85,B 0,C 180,E1 -9615.581,E2 -9615.581} C_VEL
LIN {X 0,Y 427.707,Z 588.136,A -85,B 0,C 180,E1 -9616.842,E2 -9616.842} C_VEL
LIN {X 0,Y 425.358,Z 586.652,A -85,B 0,C 180,E1 -9617.847,E2 -9617.847} C_VEL
LIN {X 0,Y 424.408,Z 585.202,A -85,B 0,C 180,E1 -9618.614,E2 -9618.614} C_VEL
LIN {X 0,Y 424.363,Z 584.633,A -85,B 0,C 180,E1 -9618.87,E2 -9618.87} C_VEL
LIN {X 0,Y 424.577,Z 580.363,A -85,B 0,C 180,E1 -9620.472,E2 -9620.472} C_VEL
LIN {X 0,Y 424.908,Z 575.278,A -85,B 0,C 180,E1 -9621.918,E2 -9621.918} C_VEL
LIN {X 0,Y 425.284,Z 568.888,A -85,B 0,C 180,E1 -9623.357,E2 -9623.357} C_VEL
LIN {X 0,Y 425.784,Z 560.906,A -85,B 0,C 180,E1 -9624.791,E2 -9624.791} C_VEL
LIN {X 0,Y 426.294,Z 552.782,A -85,B 0,C 180,E1 -9625.982,E2 -9625.982} C_VEL
LIN {X 0,Y 426.937,Z 542.875,A -85,B 0,C 180,E1 -9627.169,E2 -9627.169} C_VEL
LIN {X 0,Y 427.641,Z 531.685,A -85,B 0,C 180,E1 -9628.234,E2 -9628.234} C_VEL
LIN {X 0,Y 428.252,Z 520.728,A -85,B 0,C 180,E1 -9629.06,E2 -9629.06} C_VEL
LIN {X 0,Y 428.791,Z 508.18,A -85,B 0,C 180,E1 -9629.788,E2 -9629.788} C_VEL
LIN {X 0,Y 429.221,Z 495.944,A -85,B 0,C 180,E1 -9630.294,E2 -9630.294} C_VEL
LIN {X 0,Y 429.417,Z 483.702,A -85,B 0,C 180,E1 -9630.628,E2 -9630.628} C_VEL
LIN {X 0,Y 430.354,Z 397.899,A -85,B 0,C 180,E1 -9632.074,E2 -9632.074} C_VEL
LIN {X 0,Y 426.784,Z 380.063,A -85,B 0,C 180,E1 -9632.539,E2 -9632.539} C_VEL
LIN {X 0,Y 426.929,Z 376.866,A -85,B 0,C 180,E1 -9633.303,E2 -9633.303} C_VEL
LIN {X 0,Y 425.533,Z 368.482,A -85,B 0,C 180,E1 -9635.449,E2 -9635.449} C_VEL
LIN {X 0,Y 425.413,Z 368.493,A -85,B 0,C 180,E1 -9638.55,E2 -9638.55} C_VEL
LIN {X 0,Y 425.417,Z 368.489,A -85,B 0,C 180,E1 -9642.401,E2 -9642.401} C_VEL
LIN {X 0,Y 425.393,Z 368.492,A -85,B 0,C 180,E1 -9646.311,E2 -9646.311} C_VEL
LIN {X 0,Y 425.333,Z 368.503,A -85,B 0,C 180,E1 -9649.635,E2 -9649.635} C_VEL
LIN {X 0,Y 425.311,Z 368.509,A -85,B 0,C 180,E1 -9653.364,E2 -9653.364} C_VEL
LIN {X 0,Y 425.35,Z 368.5,A -85,B 0,C 180,E1 -9656.843,E2 -9656.843} C_VEL
LIN {X 0,Y 425.314,Z 368.504,A -85,B 0,C 180,E1 -9659.717,E2 -9659.717} C_VEL
LIN {X 0,Y 425.286,Z 368.511,A -85,B 0,C 180,E1 -9663.047,E2 -9663.047} C_VEL
LIN {X 0,Y 425.285,Z 368.506,A -85,B 0,C 180,E1 -9665.928,E2 -9665.928} C_VEL
LIN {X 0,Y 425.305,Z 368.51,A -85,B 0,C 180,E1 -9669.044,E2 -9669.044} C_VEL
LIN {X 0,Y 425.273,Z 368.51,A -85,B 0,C 180,E1 -9672.652,E2 -9672.652} C_VEL
LIN {X 0,Y 425.267,Z 368.508,A -85,B 0,C 180,E1 -9676.044,E2 -9676.044} C_VEL
LIN {X 0,Y 425.282,Z 368.508,A -85,B 0,C 180,E1 -9679.478,E2 -9679.478} C_VEL
LIN {X 0,Y 425.281,Z 368.508,A -85,B 0,C 180,E1 -9682.486,E2 -9682.486} C_VEL
LIN {X 0,Y 425.303,Z 368.503,A -85,B 0,C 180,E1 -9685.816,E2 -9685.816} C_VEL
LIN {X 0,Y 425.285,Z 368.508,A -85,B 0,C 180,E1 -9689.238,E2 -9689.238} C_VEL
LIN {X 0,Y 425.344,Z 368.501,A -85,B 0,C 180,E1 -9692.442,E2 -9692.442} C_VEL
LIN {X 0,Y 425.345,Z 368.498,A -85,B 0,C 180,E1 -9695.601,E2 -9695.601} C_VEL
LIN {X 0,Y 425.287,Z 368.512,A -85,B 0,C 180,E1 -9698.681,E2 -9698.681} C_VEL
LIN {X 0,Y 425.326,Z 368.5,A -85,B 0,C 180,E1 -9701.702,E2 -9701.702} C_VEL
LIN {X 0,Y 425.342,Z 368.506,A -85,B 0,C 180,E1 -9704.67,E2 -9704.67} C_VEL
LIN {X 0,Y 425.405,Z 368.49,A -85,B 0,C 180,E1 -9707.598,E2 -9707.598} C_VEL
LIN {X 0,Y 425.434,Z 368.487,A -85,B 0,C 180,E1 -9711.449,E2 -9711.449} C_VEL
LIN {X 0,Y 425.548,Z 368.477,A -85,B 0,C 180,E1 -9714.313,E2 -9714.313} C_VEL
LIN {X 0,Y 425.567,Z 368.473,A -85,B 0,C 180,E1 -9718.107,E2 -9718.107} C_VEL
LIN {X 0,Y 425.694,Z 368.456,A -85,B 0,C 180,E1 -9720,E2 -9720} C_VEL
LIN {X 0,Y 425.549,Z 368.476,A -85,B 0,C 180,E1 -9722.84,E2 -9722.84} C_VEL
LIN {X 0,Y 425.521,Z 368.481,A -85,B 0,C 180,E1 -9726.639,E2 -9726.639} C_VEL
LIN {X 0,Y 425.393,Z 368.492,A -85,B 0,C 180,E1 -9729.509,E2 -9729.509} C_VEL
LIN {X 0,Y 425.385,Z 368.495,A -85,B 0,C 180,E1 -9732.904,E2 -9732.904} C_VEL
LIN {X 0,Y 425.361,Z 368.5,A -85,B 0,C 180,E1 -9736.609,E2 -9736.609} C_VEL
LIN {X 0,Y 425.32,Z 368.502,A -85,B 0,C 180,E1 -9739.636,E2 -9739.636} C_VEL
LIN {X 0,Y 425.299,Z 368.504,A -85,B 0,C 180,E1 -9743.365,E2 -9743.365} C_VEL
LIN {X 0,Y 425.341,Z 368.499,A -85,B 0,C 180,E1 -9746.845,E2 -9746.845} C_VEL
LIN {X 0,Y 425.311,Z 368.504,A -85,B 0,C 180,E1 -9749.718,E2 -9749.718} C_VEL
LIN {X 0,Y 425.276,Z 368.507,A -85,B 0,C 180,E1 -9753.049,E2 -9753.049} C_VEL
LIN {X 0,Y 425.279,Z 368.511,A -85,B 0,C 180,E1 -9755.93,E2 -9755.93} C_VEL
LIN {X 0,Y 425.308,Z 368.502,A -85,B 0,C 180,E1 -9759.047,E2 -9759.047} C_VEL
LIN {X 0,Y 425.327,Z 368.501,A -85,B 0,C 180,E1 -9762.647,E2 -9762.647} C_VEL
LIN {X 0,Y 425.29,Z 368.505,A -85,B 0,C 180,E1 -9765.282,E2 -9765.282} C_VEL
LIN {X 0,Y 425.301,Z 368.504,A -85,B 0,C 180,E1 -9768.626,E2 -9768.626} C_VEL
LIN {X 0,Y 425.323,Z 368.501,A -85,B 0,C 180,E1 -9771.105,E2 -9771.105} C_VEL
LIN {X 0,Y 425.299,Z 368.504,A -85,B 0,C 180,E1 -9774.665,E2 -9774.665} C_VEL
LIN {X 0,Y 425.271,Z 368.512,A -85,B 0,C 180,E1 -9778.074,E2 -9778.074} C_VEL
LIN {X 0,Y 425.337,Z 368.507,A -85,B 0,C 180,E1 -9781.369,E2 -9781.369} C_VEL
LIN {X 0,Y 425.422,Z 368.615,A -85,B 0,C 180,E1 -9782.214,E2 -9782.214} C_VEL
LIN {X 0,Y 428.069,Z 382.268,A -85,B 0,C 180,E1 -9784.992,E2 -9784.992} C_VEL
LIN {X 0,Y 428.159,Z 386.337,A -85,B 0,C 180,E1 -9785.773,E2 -9785.773} C_VEL
LIN {X 0,Y 427.202,Z 402.472,A -85,B 0,C 180,E1 -9788.782,E2 -9788.782} C_VEL
LIN {X 0,Y 426.386,Z 417.015,A -85,B 0,C 180,E1 -9791.463,E2 -9791.463} C_VEL
LIN {X 0,Y 430.067,Z 443.216,A -85,B 0,C 180,E1 -9792.054,E2 -9792.054} C_VEL
LIN {X 0,Y 429.217,Z 526.17,A -85,B 0,C 180,E1 -9793.472,E2 -9793.472} C_VEL
LIN {X 0,Y 428.684,Z 540.021,A -85,B 0,C 180,E1 -9793.909,E2 -9793.909} C_VEL
LIN {X 0,Y 428.092,Z 552.97,A -85,B 0,C 180,E1 -9794.528,E2 -9794.528} C_VEL
LIN {X 0,Y 427.32,Z 565.566,A -85,B 0,C 180,E1 -9795.353,E2 -9795.353} C_VEL
LIN {X 0,Y 426.649,Z 577.101,A -85,B 0,C 180,E1 -9796.331,E2 -9796.331} C_VEL
LIN {X 0,Y 426.061,Z 586.923,A -85,B 0,C 180,E1 -9797.376,E2 -9797.376} C_VEL
LIN {X 0,Y 425.491,Z 596.069,A -85,B 0,C 180,E1 -9798.568,E2 -9798.568} C_VEL
LIN {X 0,Y 424.914,Z 604.986,A -85,B 0,C 180,E1 -9799.999,E2 -9799.999} C_VEL
LIN {X 0,Y 424.567,Z 612.131,A -85,B 0,C 180,E1 -9801.432,E2 -9801.432} C_VEL
LIN {X 0,Y 424.339,Z 617.828,A -85,B 0,C 180,E1 -9802.865,E2 -9802.865} C_VEL
LIN {X 0,Y 424.195,Z 622.307,A -85,B 0,C 180,E1 -9804.295,E2 -9804.295} C_VEL
LIN {X 0,Y 424.21,Z 624.672,A -85,B 0,C 180,E1 -9805.249,E2 -9805.249} C_VEL
LIN {X 0,Y 424.114,Z 626.595,A -85,B 0,C 180,E1 -9806.2,E2 -9806.2} C_VEL
LIN {X 0,Y 424.192,Z 628.085,A -85,B 0,C 180,E1 -9807.151,E2 -9807.151} C_VEL
LIN {X 0,Y 424.165,Z 629.125,A -85,B 0,C 180,E1 -9808.101,E2 -9808.101} C_VEL
LIN {X 0,Y 424.135,Z 630.029,A -85,B 0,C 180,E1 -9810,E2 -9810} C_VEL
LIN {X 0,Y 424.135,Z 629.88,A -85,B 0,C 180,E1 -9810.949,E2 -9810.949} C_VEL
LIN {X 0,Y 424.165,Z 629.303,A -85,B 0,C 180,E1 -9811.899,E2 -9811.899} C_VEL
LIN {X 0,Y 424.176,Z 628.335,A -85,B 0,C 180,E1 -9812.849,E2 -9812.849} C_VEL
LIN {X 0,Y 424.11,Z 626.967,A -85,B 0,C 180,E1 -9813.801,E2 -9813.801} C_VEL
LIN {X 0,Y 424.213,Z 624.092,A -85,B 0,C 180,E1 -9815.228,E2 -9815.228} C_VEL
LIN {X 0,Y 424.299,Z 620.188,A -85,B 0,C 180,E1 -9816.658,E2 -9816.658} C_VEL
LIN {X 0,Y 424.507,Z 615.16,A -85,B 0,C 180,E1 -9818.09,E2 -9818.09} C_VEL
LIN {X 0,Y 424.816,Z 608.859,A -85,B 0,C 180,E1 -9819.522,E2 -9819.522} C_VEL
LIN {X 0,Y 425.35,Z 600.998,A -85,B 0,C 180,E1 -9820.953,E2 -9820.953} C_VEL
LIN {X 0,Y 426.11,Z 591.209,A -85,B 0,C 180,E1 -9822.381,E2 -9822.381} C_VEL
LIN {X 0,Y 426.796,Z 580.621,A -85,B 0,C 180,E1 -9823.619,E2 -9823.619} C_VEL
LIN {X 0,Y 427.582,Z 569.664,A -85,B 0,C 180,E1 -9824.638,E2 -9824.638} C_VEL
LIN {X 0,Y 428.301,Z 558.475,A -85,B 0,C 180,E1 -9825.464,E2 -9825.464} C_VEL
LIN {X 0,Y 429.099,Z 545.946,A -85,B 0,C 180,E1 -9826.166,E2 -9826.166} C_VEL
LIN {X 0,Y 429.687,Z 532.586,A -85,B 0,C 180,E1 -9826.693,E2 -9826.693} C_VEL
LIN {X 0,Y 430.057,Z 519.495,A -85,B 0,C 180,E1 -9827.015,E2 -9827.015} C_VEL
LIN {X 0,Y 430.905,Z 442.619,A -85,B 0,C 180,E1 -9828.323,E2 -9828.323} C_VEL
LIN {X 0,Y 427.471,Z 420.596,A -85,B 0,C 180,E1 -9828.883,E2 -9828.883} C_VEL
LIN {X 0,Y 426.754,Z 416.451,A -85,B 0,C 180,E1 -9829.014,E2 -9829.014} C_VEL
LIN {X 0,Y 427.919,Z 398.312,A -85,B 0,C 180,E1 -9832.448,E2 -9832.448} C_VEL
LIN {X 0,Y 428.766,Z 385.265,A -85,B 0,C 180,E1 -9834.965,E2 -9834.965} C_VEL
LIN {X 0,Y 426.825,Z 374.642,A -85,B 0,C 180,E1 -9837.233,E2 -9837.233} C_VEL
LIN {X 0,Y 425.337,Z 368.507,A -85,B 0,C 180,E1 -9838.631,E2 -9838.631} C_VEL
LIN {X 0,Y 425.271,Z 368.513,A -85,B 0,C 180,E1 -9841.926,E2 -9841.926} C_VEL
LIN {X 0,Y 425.299,Z 368.506,A -85,B 0,C 180,E1 -9845.335,E2 -9845.335} C_VEL
LIN {X 0,Y 425.312,Z 368.502,A -85,B 0,C 180,E1 -9849.046,E2 -9849.046} C_VEL
LIN {X 0,Y 425.311,Z 368.501,A -85,B 0,C 180,E1 -9851.961,E2 -9851.961} C_VEL
LIN {X 0,Y 425.309,Z 368.505,A -85,B 0,C 180,E1 -9855.278,E2 -9855.278} C_VEL
LIN {X 0,Y 425.305,Z 368.505,A -85,B 0,C 180,E1 -9858.625,E2 -9858.625} C_VEL
LIN {X 0,Y 425.319,Z 368.502,A -85,B 0,C 180,E1 -9861.104,E2 -9861.104} C_VEL
LIN {X 0,Y 425.294,Z 368.506,A -85,B 0,C 180,E1 -9864.664,E2 -9864.664} C_VEL
LIN {X 0,Y 425.26,Z 368.513,A -85,B 0,C 180,E1 -9868.073,E2 -9868.073} C_VEL
LIN {X 0,Y 425.331,Z 368.501,A -85,B 0,C 180,E1 -9871.368,E2 -9871.368} C_VEL
LIN {X 0,Y 425.288,Z 368.503,A -85,B 0,C 180,E1 -9874.554,E2 -9874.554} C_VEL
LIN {X 0,Y 425.28,Z 368.507,A -85,B 0,C 180,E1 -9877.661,E2 -9877.661} C_VEL
LIN {X 0,Y 425.354,Z 368.498,A -85,B 0,C 180,E1 -9880.704,E2 -9880.704} C_VEL
LIN {X 0,Y 425.39,Z 368.495,A -85,B 0,C 180,E1 -9883.688,E2 -9883.688} C_VEL
LIN {X 0,Y 425.403,Z 368.49,A -85,B 0,C 180,E1 -9887.598,E2 -9887.598} C_VEL
LIN {X 0,Y 425.434,Z 368.488,A -85,B 0,C 180,E1 -9891.45,E2 -9891.45} C_VEL
LIN {X 0,Y 425.546,Z 368.474,A -85,B 0,C 180,E1 -9894.313,E2 -9894.313} C_VEL
LIN {X 0,Y 425.567,Z 368.468,A -85,B 0,C 180,E1 -9898.107,E2 -9898.107} C_VEL
LIN {X 0,Y 425.696,Z 368.456,A -85,B 0,C 180,E1 -9900,E2 -9900} C_VEL
LIN {X 0,Y 425.551,Z 368.469,A -85,B 0,C 180,E1 -9902.84,E2 -9902.84} C_VEL
LIN {X 0,Y 425.523,Z 368.476,A -85,B 0,C 180,E1 -9906.651,E2 -9906.651} C_VEL
LIN {X 0,Y 425.394,Z 368.497,A -85,B 0,C 180,E1 -9909.51,E2 -9909.51} C_VEL
LIN {X 0,Y 425.386,Z 368.492,A -85,B 0,C 180,E1 -9912.905,E2 -9912.905} C_VEL
LIN {X 0,Y 425.354,Z 368.495,A -85,B 0,C 180,E1 -9916.606,E2 -9916.606} C_VEL
LIN {X 0,Y 425.355,Z 368.495,A -85,B 0,C 180,E1 -9919.649,E2 -9919.649} C_VEL
LIN {X 0,Y 425.304,Z 368.503,A -85,B 0,C 180,E1 -9923.366,E2 -9923.366} C_VEL
LIN {X 0,Y 425.343,Z 368.503,A -85,B 0,C 180,E1 -9926.845,E2 -9926.845} C_VEL
LIN {X 0,Y 425.285,Z 368.506,A -85,B 0,C 180,E1 -9929.72,E2 -9929.72} C_VEL
LIN {X 0,Y 425.277,Z 368.506,A -85,B 0,C 180,E1 -9933.049,E2 -9933.049} C_VEL
LIN {X 0,Y 425.281,Z 368.507,A -85,B 0,C 180,E1 -9935.93,E2 -9935.93} C_VEL
LIN {X 0,Y 425.308,Z 368.508,A -85,B 0,C 180,E1 -9939.047,E2 -9939.047} C_VEL
LIN {X 0,Y 425.329,Z 368.5,A -85,B 0,C 180,E1 -9942.647,E2 -9942.647} C_VEL
LIN {X 0,Y 425.267,Z 368.511,A -85,B 0,C 180,E1 -9946.046,E2 -9946.046} C_VEL
LIN {X 0,Y 425.284,Z 368.511,A -85,B 0,C 180,E1 -9949.48,E2 -9949.48} C_VEL
LIN {X 0,Y 425.355,Z 368.712,A -85,B 0,C 180,E1 -9951.94,E2 -9951.94} C_VEL
LIN {X 0,Y 427.261,Z 378.66,A -85,B 0,C 180,E1 -9954.603,E2 -9954.603} C_VEL
LIN {X 0,Y 427.28,Z 380.565,A -85,B 0,C 180,E1 -9955.081,E2 -9955.081} C_VEL
LIN {X 0,Y 431.376,Z 398.163,A -85,B 0,C 180,E1 -9955.616,E2 -9955.616} C_VEL
LIN {X 0,Y 430.257,Z 486.709,A -85,B 0,C 180,E1 -9957.139,E2 -9957.139} C_VEL
LIN {X 0,Y 429.857,Z 500.051,A -85,B 0,C 180,E1 -9957.557,E2 -9957.557} C_VEL
LIN {X 0,Y 429.373,Z 512.984,A -85,B 0,C 180,E1 -9958.167,E2 -9958.167} C_VEL
LIN {X 0,Y 428.784,Z 524.634,A -85,B 0,C 180,E1 -9958.916,E2 -9958.916} C_VEL
LIN {X 0,Y 428.113,Z 535.562,A -85,B 0,C 180,E1 -9959.819,E2 -9959.819} C_VEL
LIN {X 0,Y 427.353,Z 545.761,A -85,B 0,C 180,E1 -9960.866,E2 -9960.866} C_VEL
LIN {X 0,Y 426.642,Z 554.759,A -85,B 0,C 180,E1 -9962,E2 -9962} C_VEL
LIN {X 0,Y 426.076,Z 562.766,A -85,B 0,C 180,E1 -9963.235,E2 -9963.235} C_VEL
LIN {X 0,Y 425.394,Z 570.883,A -85,B 0,C 180,E1 -9964.793,E2 -9964.793} C_VEL
LIN {X 0,Y 425.028,Z 576.356,A -85,B 0,C 180,E1 -9966.102,E2 -9966.102} C_VEL
LIN {X 0,Y 424.677,Z 581.426,A -85,B 0,C 180,E1 -9967.628,E2 -9967.628} C_VEL
LIN {X 0,Y 424.419,Z 585.23,A -85,B 0,C 180,E1 -9969.145,E2 -9969.145} C_VEL
LIN {X 0,Y 424.207,Z 588.113,A -85,B 0,C 180,E1 -9970.795,E2 -9970.795} C_VEL
LIN {X 0,Y 424.129,Z 589.106,A -85,B 0,C 180,E1 -9971.649,E2 -9971.649} C_VEL
LIN {X 0,Y 424.051,Z 589.835,A -85,B 0,C 180,E1 -9972.644,E2 -9972.644} C_VEL
LIN {X 0,Y 424.066,Z 590.176,A -85,B 0,C 180,E1 -9973.995,E2 -9973.995} C_VEL
LIN {X 0,Y 424.061,Z 589.519,A -85,B 0,C 180,E1 -9975.606,E2 -9975.606} C_VEL
LIN {X 0,Y 424.125,Z 588.555,A -85,B 0,C 180,E1 -9976.586,E2 -9976.586} C_VEL
LIN {X 0,Y 424.256,Z 586.814,A -85,B 0,C 180,E1 -9977.788,E2 -9977.788} C_VEL
LIN {X 0,Y 424.363,Z 584.633,A -85,B 0,C 180,E1 -9978.87,E2 -9978.87} C_VEL
LIN {X 0,Y 423.813,Z 582.858,A -85,B 0,C 180,E1 -9979.629,E2 -9979.629} C_VEL
LIN {X 0,Y 421.143,Z 579.564,A -85,B 0,C 180,E1 -9980.847,E2 -9980.847} C_VEL
LIN {X 0,Y 418.513,Z 575.546,A -85,B 0,C 180,E1 -9982.036,E2 -9982.036} C_VEL
LIN {X 0,Y 418.033,Z 572.633,A -85,B 0,C 180,E1 -9982.74,E2 -9982.74} C_VEL
LIN {X 0,Y 418.498,Z 565.397,A -85,B 0,C 180,E1 -9984.217,E2 -9984.217} C_VEL
LIN {X 0,Y 419.086,Z 556.492,A -85,B 0,C 180,E1 -9985.672,E2 -9985.672} C_VEL
LIN {X 0,Y 419.685,Z 547.361,A -85,B 0,C 180,E1 -9986.88,E2 -9986.88} C_VEL
LIN {X 0,Y 420.39,Z 537.186,A -85,B 0,C 180,E1 -9987.964,E2 -9987.964} C_VEL
LIN {X 0,Y 421.048,Z 525.922,A -85,B 0,C 180,E1 -9988.924,E2 -9988.924} C_VEL
LIN {X 0,Y 421.689,Z 513.654,A -85,B 0,C 180,E1 -9989.737,E2 -9989.737} C_VEL
LIN {X 0,Y 422.122,Z 500.955,A -85,B 0,C 180,E1 -9990.352,E2 -9990.352} C_VEL
LIN {X 0,Y 422.466,Z 487.22,A -85,B 0,C 180,E1 -9990.796,E2 -9990.796} C_VEL
LIN {X 0,Y 423.544,Z 398.747,A -85,B 0,C 180,E1 -9992.327,E2 -9992.327} C_VEL
LIN {X 0,Y 419.85,Z 380.332,A -85,B 0,C 180,E1 -9992.824,E2 -9992.824} C_VEL
LIN {X 0,Y 419.95,Z 378.138,A -85,B 0,C 180,E1 -9993.358,E2 -9993.358} C_VEL
LIN {X 0,Y 418.513,Z 369.357,A -85,B 0,C 180,E1 -9995.601,E2 -9995.601} C_VEL
LIN {X 0,Y 418.383,Z 369.37,A -85,B 0,C 180,E1 -9998.695,E2 -9998.695} C_VEL
LIN {X 0,Y 418.321,Z 369.377,A -85,B 0,C 180,E1 -10001.631,E2 -10001.631} C_VEL
LIN {X 0,Y 418.309,Z 369.375,A -85,B 0,C 180,E1 -10004.596,E2 -10004.596} C_VEL
LIN {X 0,Y 418.292,Z 369.381,A -85,B 0,C 180,E1 -10007.603,E2 -10007.603} C_VEL
LIN {X 0,Y 418.254,Z 369.382,A -85,B 0,C 180,E1 -10010.662,E2 -10010.662} C_VEL
LIN {X 0,Y 418.292,Z 369.378,A -85,B 0,C 180,E1 -10013.78,E2 -10013.78} C_VEL
LIN {X 0,Y 418.312,Z 369.379,A -85,B 0,C 180,E1 -10017.07,E2 -10017.07} C_VEL
LIN {X 0,Y 418.26,Z 369.38,A -85,B 0,C 180,E1 -10020.27,E2 -10020.27} C_VEL
LIN {X 0,Y 418.251,Z 369.383,A -85,B 0,C 180,E1 -10023.676,E2 -10023.676} C_VEL
LIN {X 0,Y 418.246,Z 369.388,A -85,B 0,C 180,E1 -10027.222,E2 -10027.222} C_VEL
LIN {X 0,Y 418.256,Z 369.382,A -85,B 0,C 180,E1 -10029.68,E2 -10029.68} C_VEL
LIN {X 0,Y 418.228,Z 369.385,A -85,B 0,C 180,E1 -10032.32,E2 -10032.32} C_VEL
LIN {X 0,Y 418.238,Z 369.39,A -85,B 0,C 180,E1 -10035.108,E2 -10035.108} C_VEL
LIN {X 0,Y 418.24,Z 369.383,A -85,B 0,C 180,E1 -10037.766,E2 -10037.766} C_VEL
LIN {X 0,Y 418.258,Z 369.384,A -85,B 0,C 180,E1 -10040.617,E2 -10040.617} C_VEL
LIN {X 0,Y 418.242,Z 369.383,A -85,B 0,C 180,E1 -10043.975,E2 -10043.975} C_VEL
LIN {X 0,Y 418.253,Z 369.386,A -85,B 0,C 180,E1 -10047.155,E2 -10047.155} C_VEL
LIN {X 0,Y 418.263,Z 369.387,A -85,B 0,C 180,E1 -10050.895,E2 -10050.895} C_VEL
LIN {X 0,Y 418.265,Z 369.38,A -85,B 0,C 180,E1 -10054.095,E2 -10054.095} C_VEL
LIN {X 0,Y 418.232,Z 369.386,A -85,B 0,C 180,E1 -10057.263,E2 -10057.263} C_VEL
LIN {X 0,Y 418.276,Z 369.381,A -85,B 0,C 180,E1 -10060.363,E2 -10060.363} C_VEL
LIN {X 0,Y 418.309,Z 369.375,A -85,B 0,C 180,E1 -10063.404,E2 -10063.404} C_VEL
LIN {X 0,Y 418.339,Z 369.374,A -85,B 0,C 180,E1 -10066.998,E2 -10066.998} C_VEL
LIN {X 0,Y 418.334,Z 369.375,A -85,B 0,C 180,E1 -10070.328,E2 -10070.328} C_VEL
LIN {X 0,Y 418.485,Z 369.353,A -85,B 0,C 180,E1 -10073.249,E2 -10073.249} C_VEL
LIN {X 0,Y 418.335,Z 369.372,A -85,B 0,C 180,E1 -10075.181,E2 -10075.181} C_VEL
LIN {X 0,Y 418.536,Z 369.348,A -85,B 0,C 180,E1 -10078.075,E2 -10078.075} C_VEL
LIN {X 0,Y 418.663,Z 369.332,A -85,B 0,C 180,E1 -10080,E2 -10080} C_VEL
LIN {X 0,Y 418.503,Z 369.353,A -85,B 0,C 180,E1 -10082.888,E2 -10082.888} C_VEL
LIN {X 0,Y 418.484,Z 369.356,A -85,B 0,C 180,E1 -10086.751,E2 -10086.751} C_VEL
LIN {X 0,Y 418.333,Z 369.372,A -85,B 0,C 180,E1 -10089.671,E2 -10089.671} C_VEL
LIN {X 0,Y 418.338,Z 369.372,A -85,B 0,C 180,E1 -10093.001,E2 -10093.001} C_VEL
LIN {X 0,Y 418.312,Z 369.377,A -85,B 0,C 180,E1 -10096.739,E2 -10096.739} C_VEL
LIN {X 0,Y 418.262,Z 369.382,A -85,B 0,C 180,E1 -10099.79,E2 -10099.79} C_VEL
LIN {X 0,Y 418.23,Z 369.386,A -85,B 0,C 180,E1 -10102.736,E2 -10102.736} C_VEL
LIN {X 0,Y 418.263,Z 369.384,A -85,B 0,C 180,E1 -10105.904,E2 -10105.904} C_VEL
LIN {X 0,Y 418.267,Z 369.38,A -85,B 0,C 180,E1 -10109.162,E2 -10109.162} C_VEL
LIN {X 0,Y 418.251,Z 369.382,A -85,B 0,C 180,E1 -10112.845,E2 -10112.845} C_VEL
LIN {X 0,Y 418.243,Z 369.389,A -85,B 0,C 180,E1 -10116.239,E2 -10116.239} C_VEL
LIN {X 0,Y 418.261,Z 369.383,A -85,B 0,C 180,E1 -10119.681,E2 -10119.681} C_VEL
LIN {X 0,Y 418.28,Z 369.382,A -85,B 0,C 180,E1 -10122.33,E2 -10122.33} C_VEL
LIN {X 0,Y 418.247,Z 369.382,A -85,B 0,C 180,E1 -10125.112,E2 -10125.112} C_VEL
LIN {X 0,Y 418.253,Z 369.386,A -85,B 0,C 180,E1 -10127.77,E2 -10127.77} C_VEL
LIN {X 0,Y 418.267,Z 369.38,A -85,B 0,C 180,E1 -10130.617,E2 -10130.617} C_VEL
LIN {X 0,Y 418.245,Z 369.389,A -85,B 0,C 180,E1 -10133.977,E2 -10133.977} C_VEL
LIN {X 0,Y 418.259,Z 369.381,A -85,B 0,C 180,E1 -10137.156,E2 -10137.156} C_VEL
LIN {X 0,Y 418.274,Z 369.385,A -85,B 0,C 180,E1 -10140.84,E2 -10140.84} C_VEL
LIN {X 0,Y 418.4,Z 369.546,A -85,B 0,C 180,E1 -10142.006,E2 -10142.006} C_VEL
LIN {X 0,Y 421.044,Z 383.243,A -85,B 0,C 180,E1 -10144.845,E2 -10144.845} C_VEL
LIN {X 0,Y 421.231,Z 387.143,A -85,B 0,C 180,E1 -10145.611,E2 -10145.611} C_VEL
LIN {X 0,Y 420.223,Z 403.282,A -85,B 0,C 180,E1 -10148.669,E2 -10148.669} C_VEL
LIN {X 0,Y 419.411,Z 416.674,A -85,B 0,C 180,E1 -10151.182,E2 -10151.182} C_VEL
LIN {X 0,Y 423.234,Z 444.15,A -85,B 0,C 180,E1 -10151.815,E2 -10151.815} C_VEL
LIN {X 0,Y 422.348,Z 525.563,A -85,B 0,C 180,E1 -10153.226,E2 -10153.226} C_VEL
LIN {X 0,Y 421.851,Z 538.753,A -85,B 0,C 180,E1 -10153.641,E2 -10153.641} C_VEL
LIN {X 0,Y 421.261,Z 550.905,A -85,B 0,C 180,E1 -10154.208,E2 -10154.208} C_VEL
LIN {X 0,Y 420.541,Z 563.174,A -85,B 0,C 180,E1 -10154.988,E2 -10154.988} C_VEL
LIN {X 0,Y 419.819,Z 574.813,A -85,B 0,C 180,E1 -10155.953,E2 -10155.953} C_VEL
LIN {X 0,Y 419.178,Z 585.289,A -85,B 0,C 180,E1 -10157.042,E2 -10157.042} C_VEL
LIN {X 0,Y 418.617,Z 593.849,A -85,B 0,C 180,E1 -10158.132,E2 -10158.132} C_VEL
LIN {X 0,Y 417.935,Z 603.1,A -85,B 0,C 180,E1 -10159.586,E2 -10159.586} C_VEL
LIN {X 0,Y 417.545,Z 610.548,A -85,B 0,C 180,E1 -10161.043,E2 -10161.043} C_VEL
LIN {X 0,Y 417.331,Z 615.604,A -85,B 0,C 180,E1 -10162.258,E2 -10162.258} C_VEL
LIN {X 0,Y 417.174,Z 620.459,A -85,B 0,C 180,E1 -10163.698,E2 -10163.698} C_VEL
LIN {X 0,Y 417.14,Z 624.269,A -85,B 0,C 180,E1 -10165.168,E2 -10165.168} C_VEL
LIN {X 0,Y 417.028,Z 626.203,A -85,B 0,C 180,E1 -10166.135,E2 -10166.135} C_VEL
LIN {X 0,Y 417.09,Z 627.713,A -85,B 0,C 180,E1 -10167.103,E2 -10167.103} C_VEL
LIN {X 0,Y 417.091,Z 628.766,A -85,B 0,C 180,E1 -10168.069,E2 -10168.069} C_VEL
LIN {X 0,Y 417.052,Z 629.689,A -85,B 0,C 180,E1 -10170,E2 -10170} C_VEL
LIN {X 0,Y 417.055,Z 629.558,A -85,B 0,C 180,E1 -10170.966,E2 -10170.966} C_VEL
LIN {X 0,Y 417.091,Z 628.994,A -85,B 0,C 180,E1 -10171.931,E2 -10171.931} C_VEL
LIN {X 0,Y 417.072,Z 628.034,A -85,B 0,C 180,E1 -10172.898,E2 -10172.898} C_VEL
LIN {X 0,Y 417.024,Z 626.677,A -85,B 0,C 180,E1 -10173.865,E2 -10173.865} C_VEL
LIN {X 0,Y 417.127,Z 623.822,A -85,B 0,C 180,E1 -10175.317,E2 -10175.317} C_VEL
LIN {X 0,Y 417.231,Z 619.939,A -85,B 0,C 180,E1 -10176.771,E2 -10176.771} C_VEL
LIN {X 0,Y 417.447,Z 614.939,A -85,B 0,C 180,E1 -10178.227,E2 -10178.227} C_VEL
LIN {X 0,Y 417.784,Z 608.673,A -85,B 0,C 180,E1 -10179.684,E2 -10179.684} C_VEL
LIN {X 0,Y 418.36,Z 600.874,A -85,B 0,C 180,E1 -10181.139,E2 -10181.139} C_VEL
LIN {X 0,Y 419.16,Z 591.142,A -85,B 0,C 180,E1 -10182.589,E2 -10182.589} C_VEL
LIN {X 0,Y 419.814,Z 581.75,A -85,B 0,C 180,E1 -10183.728,E2 -10183.728} C_VEL
LIN {X 0,Y 420.594,Z 571.194,A -85,B 0,C 180,E1 -10184.763,E2 -10184.763} C_VEL
LIN {X 0,Y 421.48,Z 558.688,A -85,B 0,C 180,E1 -10185.721,E2 -10185.721} C_VEL
LIN {X 0,Y 422.322,Z 546.391,A -85,B 0,C 180,E1 -10186.433,E2 -10186.433} C_VEL
LIN {X 0,Y 422.947,Z 533.386,A -85,B 0,C 180,E1 -10186.967,E2 -10186.967} C_VEL
LIN {X 0,Y 423.355,Z 519.544,A -85,B 0,C 180,E1 -10187.324,E2 -10187.324} C_VEL
LIN {X 0,Y 424.237,Z 443.479,A -85,B 0,C 180,E1 -10188.64,E2 -10188.64} C_VEL
LIN {X 0,Y 420.864,Z 421.755,A -85,B 0,C 180,E1 -10189.208,E2 -10189.208} C_VEL
LIN {X 0,Y 419.865,Z 416.195,A -85,B 0,C 180,E1 -10189.364,E2 -10189.364} C_VEL
LIN {X 0,Y 421.1,Z 398.409,A -85,B 0,C 180,E1 -10192.798,E2 -10192.798} C_VEL
LIN {X 0,Y 421.931,Z 387.822,A -85,B 0,C 180,E1 -10194.871,E2 -10194.871} C_VEL
